KUKA KRL program: EPS_2_25369_MH2A_A_20251215023754.src

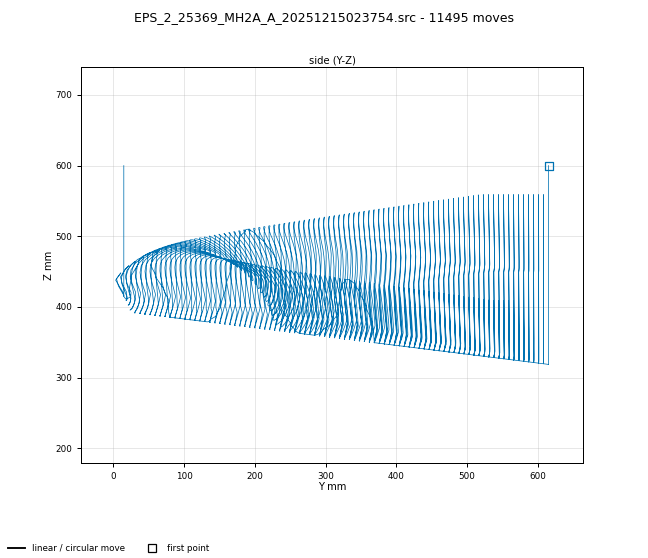
[picture p0: tool path of EPS_2_25369_MH2A_A_20251215023754.src, 11495 of 11497 moves have a stored position in this frame; points joined in program order, loops and branches not executed]
&ACCESS RVP
&REL 4
&COMMENT QRS 19112012
&PARAM EDITMASK = *
DEF PART()
EXT BAS (BAS_COMMAND :IN,REAL :IN )
INT I
BAS (#INITMOV,0 )

;KUKA QRS Post kuka4.cps  Date:22-06-2017 !

File_ID=2955

QRS_PRE_INIT()

;Init var - Until changes are made in qrs_pre_init
Outlet_Square_prg=0
Inlet_1_Square_prg=0
Inlet_2_Square_prg=0
Inlet_3_Square_prg=0
Inlet_4_Square_prg=0
Inlet_5_Square_prg=0

Outlet_1={X 0.000, Y 520.860, Z 458.500, B 0.000, E1 0.000 }
Inlet_1={X 0.000, Y 535.350, Z 258.500, B 0.000, E1 242.000 }
Outlet_1_type=201
Inlet_1_type=201
;QRS#1=Sidecore dimensions
;QRS#2=200-8" PVC SDR 35
;QRS#3=200-8" PVC SDR 35
;QRS#4=
;QRS#5=
;QRS#6=
;QRS#7=
;QRS#8=
;QRS#9=12-08 PSX
;QRS#10=12-08 PSX
;QRS#11=
;QRS#12=
;QRS#13=
;QRS#14=
;QRS#15=
;QRS#16=1220x127x838 2,75'
;QRS#17=EPS Height
;QRS#18=559
;QRS#19=*
;QRS#20= UPDATED VERSION 22-06-2017
;QRS#21=*
Outlet_Square=0100
Inlet_1_Square=0100
Inlet_2_Square=0
Inlet_3_Square=0
Inlet_4_Square=0
Inlet_5_Square=0
Mill_Square=1
Outlet_Square_Prg=204
Inlet_1_Square_prg=204

QRS_INIT()

$ADVANCE=5

; T1
PTP {E1 173.589,E2 173.589}
PTP {X 0,Y 615.517,A -85,B 0,C 180,E1 173.589,E2 173.589,E3 0,E4 0,E5 0,E6 0}
QRS_SPEED_INIT()
LIN {X 0,Y 615.517,Z 600,A -85,B 0,C 180,E1 173.589,E2 173.589,E3 0,E4 0,E5 0,E6 0} C_VEL
LIN {X 0,Y 615.517,Z 328.868,A -85,B 0,C 180,E1 173.589,E2 173.589} C_VEL
LIN {X 0,Y 615.517,Z 320.697,A -85,B 0,C 180,E1 173.589,E2 173.589} C_VEL
LIN {X 0,Y 615.495,Z 318.697,A -85,B 0,C 180,E1 173.403,E2 173.403} C_VEL
LIN {X 0,Y 615.469,Z 318.691,A -85,B 0,C 180,E1 170.801,E2 170.801} C_VEL
LIN {X 0,Y 615.46,Z 318.69,A -85,B 0,C 180,E1 168.139,E2 168.139} C_VEL
LIN {X 0,Y 615.493,Z 318.7,A -85,B 0,C 180,E1 165.451,E2 165.451} C_VEL
LIN {X 0,Y 615.461,Z 318.69,A -85,B 0,C 180,E1 162.729,E2 162.729} C_VEL
LIN {X 0,Y 615.458,Z 318.69,A -85,B 0,C 180,E1 160.661,E2 160.661} C_VEL
LIN {X 0,Y 615.457,Z 318.689,A -85,B 0,C 180,E1 158.567,E2 158.567} C_VEL
LIN {X 0,Y 615.486,Z 318.689,A -85,B 0,C 180,E1 155.989,E2 155.989} C_VEL
LIN {X 0,Y 615.489,Z 318.702,A -85,B 0,C 180,E1 153.556,E2 153.556} C_VEL
LIN {X 0,Y 615.491,Z 318.693,A -85,B 0,C 180,E1 151.342,E2 151.342} C_VEL
LIN {X 0,Y 615.465,Z 318.689,A -85,B 0,C 180,E1 148.915,E2 148.915} C_VEL
LIN {X 0,Y 615.466,Z 318.688,A -85,B 0,C 180,E1 146.467,E2 146.467} C_VEL
LIN {X 0,Y 615.494,Z 318.697,A -85,B 0,C 180,E1 143.576,E2 143.576} C_VEL
LIN {X 0,Y 615.464,Z 318.689,A -85,B 0,C 180,E1 140.939,E2 140.939} C_VEL
LIN {X 0,Y 615.471,Z 318.687,A -85,B 0,C 180,E1 138.525,E2 138.525} C_VEL
LIN {X 0,Y 615.499,Z 318.699,A -85,B 0,C 180,E1 135.851,E2 135.851} C_VEL
LIN {X 0,Y 615.467,Z 318.688,A -85,B 0,C 180,E1 133.045,E2 133.045} C_VEL
LIN {X 0,Y 615.476,Z 318.687,A -85,B 0,C 180,E1 130.606,E2 130.606} C_VEL
LIN {X 0,Y 615.491,Z 318.699,A -85,B 0,C 180,E1 128.012,E2 128.012} C_VEL
LIN {X 0,Y 615.497,Z 318.689,A -85,B 0,C 180,E1 125.614,E2 125.614} C_VEL
LIN {X 0,Y 615.472,Z 318.687,A -85,B 0,C 180,E1 123.236,E2 123.236} C_VEL
LIN {X 0,Y 615.471,Z 318.686,A -85,B 0,C 180,E1 120.92,E2 120.92} C_VEL
LIN {X 0,Y 615.495,Z 318.688,A -85,B 0,C 180,E1 118.451,E2 118.451} C_VEL
LIN {X 0,Y 615.486,Z 318.687,A -85,B 0,C 180,E1 115.568,E2 115.568} C_VEL
LIN {X 0,Y 615.479,Z 318.686,A -85,B 0,C 180,E1 112.844,E2 112.844} C_VEL
LIN {X 0,Y 615.497,Z 318.695,A -85,B 0,C 180,E1 110.032,E2 110.032} C_VEL
LIN {X 0,Y 615.473,Z 318.686,A -85,B 0,C 180,E1 107.27,E2 107.27} C_VEL
LIN {X 0,Y 615.494,Z 318.691,A -85,B 0,C 180,E1 104.549,E2 104.549} C_VEL
LIN {X 0,Y 615.49,Z 318.689,A -85,B 0,C 180,E1 101.86,E2 101.86} C_VEL
LIN {X 0,Y 615.478,Z 318.685,A -85,B 0,C 180,E1 99.199,E2 99.199} C_VEL
LIN {X 0,Y 615.494,Z 318.694,A -85,B 0,C 180,E1 96.556,E2 96.556} C_VEL
LIN {X 0,Y 615.489,Z 318.688,A -85,B 0,C 180,E1 93.928,E2 93.928} C_VEL
LIN {X 0,Y 615.48,Z 318.684,A -85,B 0,C 180,E1 91.309,E2 91.309} C_VEL
LIN {X 0,Y 615.494,Z 318.694,A -85,B 0,C 180,E1 88.691,E2 88.691} C_VEL
LIN {X 0,Y 615.491,Z 318.688,A -85,B 0,C 180,E1 86.072,E2 86.072} C_VEL
LIN {X 0,Y 615.48,Z 318.684,A -85,B 0,C 180,E1 83.43,E2 83.43} C_VEL
LIN {X 0,Y 615.49,Z 318.695,A -85,B 0,C 180,E1 80.801,E2 80.801} C_VEL
LIN {X 0,Y 615.49,Z 318.687,A -85,B 0,C 180,E1 78.14,E2 78.14} C_VEL
LIN {X 0,Y 615.484,Z 318.684,A -85,B 0,C 180,E1 75.451,E2 75.451} C_VEL
LIN {X 0,Y 615.498,Z 318.699,A -85,B 0,C 180,E1 72.73,E2 72.73} C_VEL
LIN {X 0,Y 615.485,Z 318.684,A -85,B 0,C 180,E1 69.968,E2 69.968} C_VEL
LIN {X 0,Y 615.491,Z 318.69,A -85,B 0,C 180,E1 67.156,E2 67.156} C_VEL
LIN {X 0,Y 615.5,Z 318.684,A -85,B 0,C 180,E1 64.286,E2 64.286} C_VEL
LIN {X 0,Y 615.493,Z 318.683,A -85,B 0,C 180,E1 61.549,E2 61.549} C_VEL
LIN {X 0,Y 615.491,Z 318.702,A -85,B 0,C 180,E1 58.914,E2 58.914} C_VEL
LIN {X 0,Y 615.491,Z 318.688,A -85,B 0,C 180,E1 56.466,E2 56.466} C_VEL
LIN {X 0,Y 615.489,Z 318.685,A -85,B 0,C 180,E1 53.576,E2 53.576} C_VEL
LIN {X 0,Y 615.492,Z 318.699,A -85,B 0,C 180,E1 50.938,E2 50.938} C_VEL
LIN {X 0,Y 615.495,Z 318.686,A -85,B 0,C 180,E1 48.528,E2 48.528} C_VEL
LIN {X 0,Y 615.493,Z 318.682,A -85,B 0,C 180,E1 45.852,E2 45.852} C_VEL
LIN {X 0,Y 615.492,Z 318.699,A -85,B 0,C 180,E1 43.049,E2 43.049} C_VEL
LIN {X 0,Y 615.495,Z 318.685,A -85,B 0,C 180,E1 40.606,E2 40.606} C_VEL
LIN {X 0,Y 615.492,Z 318.789,A -85,B 0,C 180,E1 39.236,E2 39.236} C_VEL
LIN {X 0,Y 615.494,Z 331.581,A -85,B 0,C 180,E1 38.799,E2 38.799} C_VEL
LIN {X 0,Y 615.494,Z 341.036,A -85,B 0,C 180,E1 38.38,E2 38.38} C_VEL
LIN {X 0,Y 615.496,Z 349.628,A -85,B 0,C 180,E1 37.918,E2 37.918} C_VEL
LIN {X 0,Y 615.498,Z 358.544,A -85,B 0,C 180,E1 37.338,E2 37.338} C_VEL
LIN {X 0,Y 615.499,Z 366.968,A -85,B 0,C 180,E1 36.681,E2 36.681} C_VEL
LIN {X 0,Y 615.497,Z 374.514,A -85,B 0,C 180,E1 35.984,E2 35.984} C_VEL
LIN {X 0,Y 615.498,Z 381.527,A -85,B 0,C 180,E1 35.214,E2 35.214} C_VEL
LIN {X 0,Y 615.496,Z 386.825,A -85,B 0,C 180,E1 34.532,E2 34.532} C_VEL
LIN {X 0,Y 615.491,Z 391.828,A -85,B 0,C 180,E1 33.78,E2 33.78} C_VEL
LIN {X 0,Y 615.493,Z 396.922,A -85,B 0,C 180,E1 32.846,E2 32.846} C_VEL
LIN {X 0,Y 615.492,Z 400.615,A -85,B 0,C 180,E1 32.009,E2 32.009} C_VEL
LIN {X 0,Y 615.488,Z 404.238,A -85,B 0,C 180,E1 30.92,E2 30.92} C_VEL
LIN {X 0,Y 615.493,Z 406.751,A -85,B 0,C 180,E1 29.798,E2 29.798} C_VEL
LIN {X 0,Y 615.485,Z 407.427,A -85,B 0,C 180,E1 29.406,E2 29.406} C_VEL
LIN {X 0,Y 615.497,Z 408.272,A -85,B 0,C 180,E1 28.455,E2 28.455} C_VEL
LIN {X 0,Y 615.489,Z 407.929,A -85,B 0,C 180,E1 27.048,E2 27.048} C_VEL
LIN {X 0,Y 615.489,Z 407.306,A -85,B 0,C 180,E1 26.444,E2 26.444} C_VEL
LIN {X 0,Y 615.489,Z 405.769,A -85,B 0,C 180,E1 25.572,E2 25.572} C_VEL
LIN {X 0,Y 615.496,Z 403.25,A -85,B 0,C 180,E1 24.631,E2 24.631} C_VEL
LIN {X 0,Y 615.486,Z 399.206,A -85,B 0,C 180,E1 23.556,E2 23.556} C_VEL
LIN {X 0,Y 615.498,Z 394.51,A -85,B 0,C 180,E1 22.597,E2 22.597} C_VEL
LIN {X 0,Y 615.496,Z 389.635,A -85,B 0,C 180,E1 21.783,E2 21.783} C_VEL
LIN {X 0,Y 615.496,Z 383.247,A -85,B 0,C 180,E1 20.905,E2 20.905} C_VEL
LIN {X 0,Y 615.499,Z 376.823,A -85,B 0,C 180,E1 20.165,E2 20.165} C_VEL
LIN {X 0,Y 615.499,Z 370.184,A -85,B 0,C 180,E1 19.511,E2 19.511} C_VEL
LIN {X 0,Y 615.498,Z 361.856,A -85,B 0,C 180,E1 18.818,E2 18.818} C_VEL
LIN {X 0,Y 615.497,Z 352.996,A -85,B 0,C 180,E1 18.202,E2 18.202} C_VEL
LIN {X 0,Y 615.497,Z 344.313,A -85,B 0,C 180,E1 17.699,E2 17.699} C_VEL
LIN {X 0,Y 615.498,Z 335.372,A -85,B 0,C 180,E1 17.27,E2 17.27} C_VEL
LIN {X 0,Y 615.497,Z 326.627,A -85,B 0,C 180,E1 16.928,E2 16.928} C_VEL
LIN {X 0,Y 615.497,Z 319.573,A -85,B 0,C 180,E1 16.672,E2 16.672} C_VEL
LIN {X 0,Y 615.495,Z 318.786,A -85,B 0,C 180,E1 16.512,E2 16.512} C_VEL
LIN {X 0,Y 615.463,Z 318.69,A -85,B 0,C 180,E1 13.875,E2 13.875} C_VEL
LIN {X 0,Y 615.468,Z 318.69,A -85,B 0,C 180,E1 11.193,E2 11.193} C_VEL
LIN {X 0,Y 615.496,Z 318.698,A -85,B 0,C 180,E1 8.537,E2 8.537} C_VEL
LIN {X 0,Y 615.456,Z 318.691,A -85,B 0,C 180,E1 5.899,E2 5.899} C_VEL
LIN {X 0,Y 615.467,Z 318.69,A -85,B 0,C 180,E1 3.273,E2 3.273} C_VEL
LIN {X 0,Y 615.496,Z 318.699,A -85,B 0,C 180,E1 0.654,E2 0.654} C_VEL
LIN {X 0,Y 615.455,Z 318.692,A -85,B 0,C 180,E1 -1.963,E2 -1.963} C_VEL
LIN {X 0,Y 615.452,Z 318.692,A -85,B 0,C 180,E1 -3.929,E2 -3.929} C_VEL
LIN {X 0,Y 615.454,Z 318.692,A -85,B 0,C 180,E1 -5.899,E2 -5.899} C_VEL
LIN {X 0,Y 615.451,Z 318.693,A -85,B 0,C 180,E1 -7.876,E2 -7.876} C_VEL
LIN {X 0,Y 615.451,Z 318.692,A -85,B 0,C 180,E1 -9.863,E2 -9.863} C_VEL
LIN {X 0,Y 615.449,Z 318.693,A -85,B 0,C 180,E1 -11.862,E2 -11.862} C_VEL
LIN {X 0,Y 615.445,Z 318.693,A -85,B 0,C 180,E1 -13.923,E2 -13.923} C_VEL
LIN {X 0,Y 615.472,Z 318.691,A -85,B 0,C 180,E1 -16.587,E2 -16.587} C_VEL
LIN {X 0,Y 615.479,Z 318.694,A -85,B 0,C 180,E1 -19.338,E2 -19.338} C_VEL
LIN {X 0,Y 615.461,Z 318.695,A -85,B 0,C 180,E1 -21.433,E2 -21.433} C_VEL
LIN {X 0,Y 615.452,Z 318.694,A -85,B 0,C 180,E1 -23.558,E2 -23.558} C_VEL
LIN {X 0,Y 615.441,Z 318.694,A -85,B 0,C 180,E1 -25.718,E2 -25.718} C_VEL
LIN {X 0,Y 615.438,Z 318.693,A -85,B 0,C 180,E1 -27.918,E2 -27.918} C_VEL
LIN {X 0,Y 615.492,Z 318.701,A -85,B 0,C 180,E1 -30.92,E2 -30.92} C_VEL
LIN {X 0,Y 615.442,Z 318.695,A -85,B 0,C 180,E1 -33.53,E2 -33.53} C_VEL
LIN {X 0,Y 615.435,Z 318.694,A -85,B 0,C 180,E1 -35.829,E2 -35.829} C_VEL
LIN {X 0,Y 615.445,Z 318.694,A -85,B 0,C 180,E1 -38.072,E2 -38.072} C_VEL
LIN {X 0,Y 615.491,Z 318.696,A -85,B 0,C 180,E1 -40.606,E2 -40.606} C_VEL
LIN {X 0,Y 615.446,Z 318.696,A -85,B 0,C 180,E1 -43.248,E2 -43.248} C_VEL
LIN {X 0,Y 615.445,Z 318.694,A -85,B 0,C 180,E1 -46.007,E2 -46.007} C_VEL
LIN {X 0,Y 615.469,Z 318.698,A -85,B 0,C 180,E1 -48.908,E2 -48.908} C_VEL
LIN {X 0,Y 615.446,Z 318.698,A -85,B 0,C 180,E1 -51.094,E2 -51.094} C_VEL
LIN {X 0,Y 615.427,Z 318.696,A -85,B 0,C 180,E1 -53.572,E2 -53.572} C_VEL
LIN {X 0,Y 615.495,Z 318.898,A -85,B 0,C 180,E1 -54.687,E2 -54.687} C_VEL
LIN {X 0,Y 615.497,Z 333.444,A -85,B 0,C 180,E1 -57.35,E2 -57.35} C_VEL
LIN {X 0,Y 615.496,Z 348.208,A -85,B 0,C 180,E1 -60.204,E2 -60.204} C_VEL
LIN {X 0,Y 615.465,Z 362.707,A -85,B 0,C 180,E1 -62.96,E2 -62.96} C_VEL
LIN {X 0,Y 615.477,Z 375.666,A -85,B 0,C 180,E1 -65.369,E2 -65.369} C_VEL
LIN {X 0,Y 615.496,Z 391.293,A -85,B 0,C 180,E1 -68.217,E2 -68.217} C_VEL
LIN {X 0,Y 615.462,Z 406.91,A -85,B 0,C 180,E1 -71.008,E2 -71.008} C_VEL
LIN {X 0,Y 615.462,Z 421.502,A -85,B 0,C 180,E1 -73.578,E2 -73.578} C_VEL
LIN {X 0,Y 615.488,Z 438.093,A -85,B 0,C 180,E1 -76.463,E2 -76.463} C_VEL
LIN {X 0,Y 615.485,Z 448.706,A -85,B 0,C 180,E1 -78.265,E2 -78.265} C_VEL
LIN {X 0,Y 615.482,Z 449.705,A -85,B 0,C 180,E1 -78.327,E2 -78.327} C_VEL
LIN {X 0,Y 615.47,Z 464.052,A -85,B 0,C 180,E1 -78.598,E2 -78.598} C_VEL
LIN {X 0,Y 615.474,Z 476.487,A -85,B 0,C 180,E1 -78.961,E2 -78.961} C_VEL
LIN {X 0,Y 615.494,Z 487.108,A -85,B 0,C 180,E1 -79.384,E2 -79.384} C_VEL
LIN {X 0,Y 615.497,Z 498.603,A -85,B 0,C 180,E1 -79.972,E2 -79.972} C_VEL
LIN {X 0,Y 615.499,Z 510.015,A -85,B 0,C 180,E1 -80.719,E2 -80.719} C_VEL
LIN {X 0,Y 615.498,Z 519.243,A -85,B 0,C 180,E1 -81.464,E2 -81.464} C_VEL
LIN {X 0,Y 615.499,Z 527.669,A -85,B 0,C 180,E1 -82.29,E2 -82.29} C_VEL
LIN {X 0,Y 615.498,Z 535.689,A -85,B 0,C 180,E1 -83.258,E2 -83.258} C_VEL
LIN {X 0,Y 615.499,Z 541.428,A -85,B 0,C 180,E1 -84.102,E2 -84.102} C_VEL
LIN {X 0,Y 615.495,Z 546.876,A -85,B 0,C 180,E1 -85.087,E2 -85.087} C_VEL
LIN {X 0,Y 615.497,Z 551.143,A -85,B 0,C 180,E1 -86.072,E2 -86.072} C_VEL
LIN {X 0,Y 615.494,Z 553.397,A -85,B 0,C 180,E1 -86.727,E2 -86.727} C_VEL
LIN {X 0,Y 615.496,Z 555.231,A -85,B 0,C 180,E1 -87.382,E2 -87.382} C_VEL
LIN {X 0,Y 615.5,Z 556.61,A -85,B 0,C 180,E1 -88.037,E2 -88.037} C_VEL
LIN {X 0,Y 615.496,Z 558.173,A -85,B 0,C 180,E1 -89.346,E2 -89.346} C_VEL
LIN {X 0,Y 615.494,Z 558.389,A -85,B 0,C 180,E1 -90,E2 -90} C_VEL
LIN {X 0,Y 615.495,Z 557.581,A -85,B 0,C 180,E1 -91.309,E2 -91.309} C_VEL
LIN {X 0,Y 615.5,Z 556.61,A -85,B 0,C 180,E1 -91.963,E2 -91.963} C_VEL
LIN {X 0,Y 615.496,Z 555.231,A -85,B 0,C 180,E1 -92.618,E2 -92.618} C_VEL
LIN {X 0,Y 615.495,Z 552.352,A -85,B 0,C 180,E1 -93.601,E2 -93.601} C_VEL
LIN {X 0,Y 615.497,Z 548.448,A -85,B 0,C 180,E1 -94.584,E2 -94.584} C_VEL
LIN {X 0,Y 615.499,Z 543.41,A -85,B 0,C 180,E1 -95.57,E2 -95.57} C_VEL
LIN {X 0,Y 615.497,Z 536.856,A -85,B 0,C 180,E1 -96.584,E2 -96.584} C_VEL
LIN {X 0,Y 615.497,Z 529.134,A -85,B 0,C 180,E1 -97.545,E2 -97.545} C_VEL
LIN {X 0,Y 615.498,Z 521.055,A -85,B 0,C 180,E1 -98.371,E2 -98.371} C_VEL
LIN {X 0,Y 615.499,Z 511.154,A -85,B 0,C 180,E1 -99.198,E2 -99.198} C_VEL
LIN {X 0,Y 615.498,Z 499.986,A -85,B 0,C 180,E1 -99.945,E2 -99.945} C_VEL
LIN {X 0,Y 615.497,Z 489.05,A -85,B 0,C 180,E1 -100.526,E2 -100.526} C_VEL
LIN {X 0,Y 615.476,Z 477.622,A -85,B 0,C 180,E1 -101,E2 -101} C_VEL
LIN {X 0,Y 615.469,Z 465.798,A -85,B 0,C 180,E1 -101.36,E2 -101.36} C_VEL
LIN {X 0,Y 615.48,Z 452.013,A -85,B 0,C 180,E1 -101.631,E2 -101.631} C_VEL
LIN {X 0,Y 615.484,Z 449.247,A -85,B 0,C 180,E1 -101.693,E2 -101.693} C_VEL
LIN {X 0,Y 615.491,Z 447.83,A -85,B 0,C 180,E1 -101.86,E2 -101.86} C_VEL
LIN {X 0,Y 615.489,Z 432.252,A -85,B 0,C 180,E1 -104.549,E2 -104.549} C_VEL
LIN {X 0,Y 615.492,Z 416.659,A -85,B 0,C 180,E1 -107.27,E2 -107.27} C_VEL
LIN {X 0,Y 615.477,Z 401.055,A -85,B 0,C 180,E1 -110.033,E2 -110.033} C_VEL
LIN {X 0,Y 615.474,Z 386.808,A -85,B 0,C 180,E1 -112.595,E2 -112.595} C_VEL
LIN {X 0,Y 615.488,Z 372.144,A -85,B 0,C 180,E1 -115.281,E2 -115.281} C_VEL
LIN {X 0,Y 615.473,Z 356.66,A -85,B 0,C 180,E1 -118.181,E2 -118.181} C_VEL
LIN {X 0,Y 615.464,Z 344.37,A -85,B 0,C 180,E1 -120.54,E2 -120.54} C_VEL
LIN {X 0,Y 615.489,Z 330.389,A -85,B 0,C 180,E1 -123.235,E2 -123.235} C_VEL
LIN {X 0,Y 615.495,Z 319.029,A -85,B 0,C 180,E1 -125.413,E2 -125.413} C_VEL
LIN {X 0,Y 615.468,Z 318.698,A -85,B 0,C 180,E1 -125.831,E2 -125.831} C_VEL
LIN {X 0,Y 615.442,Z 318.697,A -85,B 0,C 180,E1 -128.071,E2 -128.071} C_VEL
LIN {X 0,Y 615.431,Z 318.695,A -85,B 0,C 180,E1 -130.61,E2 -130.61} C_VEL
LIN {X 0,Y 615.494,Z 318.694,A -85,B 0,C 180,E1 -133.243,E2 -133.243} C_VEL
LIN {X 0,Y 615.443,Z 318.696,A -85,B 0,C 180,E1 -136.005,E2 -136.005} C_VEL
LIN {X 0,Y 615.436,Z 318.695,A -85,B 0,C 180,E1 -138.522,E2 -138.522} C_VEL
LIN {X 0,Y 615.487,Z 318.694,A -85,B 0,C 180,E1 -141.095,E2 -141.095} C_VEL
LIN {X 0,Y 615.472,Z 318.697,A -85,B 0,C 180,E1 -143.574,E2 -143.574} C_VEL
LIN {X 0,Y 615.441,Z 318.695,A -85,B 0,C 180,E1 -145.975,E2 -145.975} C_VEL
LIN {X 0,Y 615.438,Z 318.694,A -85,B 0,C 180,E1 -148.312,E2 -148.312} C_VEL
LIN {X 0,Y 615.454,Z 318.693,A -85,B 0,C 180,E1 -150.592,E2 -150.592} C_VEL
LIN {X 0,Y 615.467,Z 318.695,A -85,B 0,C 180,E1 -153.555,E2 -153.555} C_VEL
LIN {X 0,Y 615.44,Z 318.693,A -85,B 0,C 180,E1 -155.998,E2 -155.998} C_VEL
LIN {X 0,Y 615.442,Z 318.694,A -85,B 0,C 180,E1 -157.862,E2 -157.862} C_VEL
LIN {X 0,Y 615.439,Z 318.694,A -85,B 0,C 180,E1 -159.965,E2 -159.965} C_VEL
LIN {X 0,Y 615.488,Z 318.692,A -85,B 0,C 180,E1 -162.729,E2 -162.729} C_VEL
LIN {X 0,Y 615.467,Z 318.694,A -85,B 0,C 180,E1 -165.45,E2 -165.45} C_VEL
LIN {X 0,Y 615.463,Z 318.693,A -85,B 0,C 180,E1 -167.469,E2 -167.469} C_VEL
LIN {X 0,Y 615.461,Z 318.693,A -85,B 0,C 180,E1 -169.473,E2 -169.473} C_VEL
LIN {X 0,Y 615.457,Z 318.694,A -85,B 0,C 180,E1 -171.463,E2 -171.463} C_VEL
LIN {X 0,Y 615.461,Z 318.693,A -85,B 0,C 180,E1 -173.443,E2 -173.443} C_VEL
LIN {X 0,Y 615.458,Z 318.693,A -85,B 0,C 180,E1 -175.415,E2 -175.415} C_VEL
LIN {X 0,Y 615.463,Z 318.692,A -85,B 0,C 180,E1 -177.382,E2 -177.382} C_VEL
LIN {X 0,Y 615.455,Z 318.691,A -85,B 0,C 180,E1 -180,E2 -180} C_VEL
LIN {X 0,Y 615.495,Z 318.696,A -85,B 0,C 180,E1 -182.618,E2 -182.618} C_VEL
LIN {X 0,Y 615.468,Z 318.692,A -85,B 0,C 180,E1 -185.241,E2 -185.241} C_VEL
LIN {X 0,Y 615.495,Z 318.697,A -85,B 0,C 180,E1 -186.597,E2 -186.597} C_VEL
LIN {X 0,Y 614.802,Z 318.837,A -85,B 0,C 180,E1 -187.142,E2 -187.142} C_VEL
LIN {X 0,Y 611.956,Z 319.252,A -85,B 0,C 180,E1 -188.028,E2 -188.028} C_VEL
LIN {X 0,Y 609.563,Z 319.562,A -85,B 0,C 180,E1 -188.741,E2 -188.741} C_VEL
LIN {X 0,Y 608.529,Z 319.68,A -85,B 0,C 180,E1 -189.29,E2 -189.29} C_VEL
LIN {X 0,Y 608.439,Z 319.689,A -85,B 0,C 180,E1 -189.476,E2 -189.476} C_VEL
LIN {X 0,Y 608.444,Z 319.69,A -85,B 0,C 180,E1 -192,E2 -192} C_VEL
LIN {X 0,Y 608.471,Z 319.694,A -85,B 0,C 180,E1 -194.721,E2 -194.721} C_VEL
LIN {X 0,Y 608.431,Z 319.69,A -85,B 0,C 180,E1 -197.477,E2 -197.477} C_VEL
LIN {X 0,Y 608.434,Z 319.69,A -85,B 0,C 180,E1 -199.571,E2 -199.571} C_VEL
LIN {X 0,Y 608.454,Z 319.687,A -85,B 0,C 180,E1 -201.692,E2 -201.692} C_VEL
LIN {X 0,Y 608.45,Z 319.696,A -85,B 0,C 180,E1 -204.571,E2 -204.571} C_VEL
LIN {X 0,Y 608.436,Z 319.689,A -85,B 0,C 180,E1 -207.519,E2 -207.519} C_VEL
LIN {X 0,Y 608.464,Z 319.69,A -85,B 0,C 180,E1 -209.973,E2 -209.973} C_VEL
LIN {X 0,Y 608.448,Z 319.69,A -85,B 0,C 180,E1 -212.88,E2 -212.88} C_VEL
LIN {X 0,Y 608.431,Z 319.69,A -85,B 0,C 180,E1 -215.279,E2 -215.279} C_VEL
LIN {X 0,Y 608.469,Z 319.696,A -85,B 0,C 180,E1 -218.242,E2 -218.242} C_VEL
LIN {X 0,Y 608.433,Z 319.69,A -85,B 0,C 180,E1 -221.179,E2 -221.179} C_VEL
LIN {X 0,Y 608.475,Z 319.69,A -85,B 0,C 180,E1 -223.869,E2 -223.869} C_VEL
LIN {X 0,Y 608.465,Z 319.688,A -85,B 0,C 180,E1 -226.692,E2 -226.692} C_VEL
LIN {X 0,Y 608.443,Z 319.689,A -85,B 0,C 180,E1 -228.824,E2 -228.824} C_VEL
LIN {X 0,Y 608.468,Z 319.691,A -85,B 0,C 180,E1 -231.76,E2 -231.76} C_VEL
LIN {X 0,Y 608.443,Z 319.69,A -85,B 0,C 180,E1 -234.723,E2 -234.723} C_VEL
LIN {X 0,Y 608.467,Z 319.688,A -85,B 0,C 180,E1 -237.477,E2 -237.477} C_VEL
LIN {X 0,Y 608.48,Z 319.69,A -85,B 0,C 180,E1 -240.222,E2 -240.222} C_VEL
LIN {X 0,Y 608.467,Z 319.686,A -85,B 0,C 180,E1 -242.795,E2 -242.795} C_VEL
LIN {X 0,Y 608.453,Z 319.69,A -85,B 0,C 180,E1 -245.43,E2 -245.43} C_VEL
LIN {X 0,Y 608.467,Z 319.689,A -85,B 0,C 180,E1 -248.309,E2 -248.309} C_VEL
LIN {X 0,Y 608.456,Z 319.688,A -85,B 0,C 180,E1 -251.131,E2 -251.131} C_VEL
LIN {X 0,Y 608.467,Z 319.694,A -85,B 0,C 180,E1 -253.907,E2 -253.907} C_VEL
LIN {X 0,Y 608.459,Z 319.687,A -85,B 0,C 180,E1 -256.644,E2 -256.644} C_VEL
LIN {X 0,Y 608.47,Z 319.69,A -85,B 0,C 180,E1 -259.351,E2 -259.351} C_VEL
LIN {X 0,Y 608.481,Z 319.688,A -85,B 0,C 180,E1 -262.033,E2 -262.033} C_VEL
LIN {X 0,Y 608.461,Z 319.686,A -85,B 0,C 180,E1 -264.698,E2 -264.698} C_VEL
LIN {X 0,Y 608.484,Z 319.69,A -85,B 0,C 180,E1 -267.352,E2 -267.352} C_VEL
LIN {X 0,Y 608.481,Z 319.687,A -85,B 0,C 180,E1 -270,E2 -270} C_VEL
LIN {X 0,Y 608.472,Z 319.685,A -85,B 0,C 180,E1 -272.648,E2 -272.648} C_VEL
LIN {X 0,Y 608.473,Z 319.693,A -85,B 0,C 180,E1 -275.302,E2 -275.302} C_VEL
LIN {X 0,Y 608.481,Z 319.686,A -85,B 0,C 180,E1 -277.967,E2 -277.967} C_VEL
LIN {X 0,Y 608.463,Z 319.687,A -85,B 0,C 180,E1 -280.65,E2 -280.65} C_VEL
LIN {X 0,Y 608.472,Z 319.696,A -85,B 0,C 180,E1 -283.356,E2 -283.356} C_VEL
LIN {X 0,Y 608.461,Z 319.687,A -85,B 0,C 180,E1 -286.093,E2 -286.093} C_VEL
LIN {X 0,Y 608.459,Z 319.69,A -85,B 0,C 180,E1 -288.869,E2 -288.869} C_VEL
LIN {X 0,Y 608.472,Z 319.688,A -85,B 0,C 180,E1 -291.691,E2 -291.691} C_VEL
LIN {X 0,Y 608.455,Z 319.689,A -85,B 0,C 180,E1 -294.57,E2 -294.57} C_VEL
LIN {X 0,Y 608.485,Z 319.693,A -85,B 0,C 180,E1 -297.208,E2 -297.208} C_VEL
LIN {X 0,Y 608.469,Z 319.685,A -85,B 0,C 180,E1 -299.971,E2 -299.971} C_VEL
LIN {X 0,Y 608.467,Z 319.688,A -85,B 0,C 180,E1 -302.523,E2 -302.523} C_VEL
LIN {X 0,Y 608.451,Z 319.694,A -85,B 0,C 180,E1 -305.276,E2 -305.276} C_VEL
LIN {X 0,Y 608.471,Z 319.686,A -85,B 0,C 180,E1 -307.745,E2 -307.745} C_VEL
LIN {X 0,Y 608.478,Z 319.686,A -85,B 0,C 180,E1 -310.332,E2 -310.332} C_VEL
LIN {X 0,Y 608.479,Z 319.689,A -85,B 0,C 180,E1 -313.309,E2 -313.309} C_VEL
LIN {X 0,Y 608.472,Z 319.686,A -85,B 0,C 180,E1 -316.131,E2 -316.131} C_VEL
LIN {X 0,Y 608.46,Z 319.697,A -85,B 0,C 180,E1 -318.824,E2 -318.824} C_VEL
LIN {X 0,Y 608.488,Z 319.875,A -85,B 0,C 180,E1 -320.661,E2 -320.661} C_VEL
LIN {X 0,Y 608.513,Z 332.249,A -85,B 0,C 180,E1 -321.097,E2 -321.097} C_VEL
LIN {X 0,Y 608.506,Z 341.54,A -85,B 0,C 180,E1 -321.516,E2 -321.516} C_VEL
LIN {X 0,Y 608.498,Z 351.312,A -85,B 0,C 180,E1 -322.06,E2 -322.06} C_VEL
LIN {X 0,Y 608.491,Z 359.545,A -85,B 0,C 180,E1 -322.61,E2 -322.61} C_VEL
LIN {X 0,Y 608.471,Z 368.109,A -85,B 0,C 180,E1 -323.293,E2 -323.293} C_VEL
LIN {X 0,Y 608.473,Z 375.088,A -85,B 0,C 180,E1 -323.949,E2 -323.949} C_VEL
LIN {X 0,Y 608.462,Z 382.076,A -85,B 0,C 180,E1 -324.723,E2 -324.723} C_VEL
LIN {X 0,Y 608.461,Z 388.204,A -85,B 0,C 180,E1 -325.53,E2 -325.53} C_VEL
LIN {X 0,Y 608.457,Z 393.298,A -85,B 0,C 180,E1 -326.329,E2 -326.329} C_VEL
LIN {X 0,Y 608.428,Z 397.518,A -85,B 0,C 180,E1 -327.119,E2 -327.119} C_VEL
LIN {X 0,Y 608.423,Z 402.432,A -85,B 0,C 180,E1 -328.293,E2 -328.293} C_VEL
LIN {X 0,Y 608.443,Z 403.951,A -85,B 0,C 180,E1 -328.731,E2 -328.731} C_VEL
LIN {X 0,Y 608.425,Z 405.914,A -85,B 0,C 180,E1 -329.453,E2 -329.453} C_VEL
LIN {X 0,Y 608.442,Z 407.417,A -85,B 0,C 180,E1 -330.219,E2 -330.219} C_VEL
LIN {X 0,Y 608.421,Z 408.78,A -85,B 0,C 180,E1 -331.386,E2 -331.386} C_VEL
LIN {X 0,Y 608.42,Z 408.912,A -85,B 0,C 180,E1 -332.481,E2 -332.481} C_VEL
LIN {X 0,Y 608.42,Z 408.331,A -85,B 0,C 180,E1 -333.224,E2 -333.224} C_VEL
LIN {X 0,Y 608.421,Z 406.712,A -85,B 0,C 180,E1 -334.286,E2 -334.286} C_VEL
LIN {X 0,Y 608.425,Z 403.735,A -85,B 0,C 180,E1 -335.428,E2 -335.428} C_VEL
LIN {X 0,Y 608.443,Z 399.625,A -85,B 0,C 180,E1 -336.515,E2 -336.515} C_VEL
LIN {X 0,Y 608.447,Z 394.655,A -85,B 0,C 180,E1 -337.523,E2 -337.523} C_VEL
LIN {X 0,Y 608.462,Z 388.713,A -85,B 0,C 180,E1 -338.486,E2 -338.486} C_VEL
LIN {X 0,Y 608.472,Z 382.488,A -85,B 0,C 180,E1 -339.317,E2 -339.317} C_VEL
LIN {X 0,Y 608.465,Z 375.703,A -85,B 0,C 180,E1 -340.078,E2 -340.078} C_VEL
LIN {X 0,Y 608.467,Z 366.351,A -85,B 0,C 180,E1 -340.956,E2 -340.956} C_VEL
LIN {X 0,Y 608.515,Z 355.759,A -85,B 0,C 180,E1 -341.747,E2 -341.747} C_VEL
LIN {X 0,Y 608.499,Z 345.79,A -85,B 0,C 180,E1 -342.351,E2 -342.351} C_VEL
LIN {X 0,Y 608.513,Z 336.117,A -85,B 0,C 180,E1 -342.828,E2 -342.828} C_VEL
LIN {X 0,Y 608.541,Z 326.217,A -85,B 0,C 180,E1 -343.218,E2 -343.218} C_VEL
LIN {X 0,Y 608.552,Z 320.356,A -85,B 0,C 180,E1 -343.439,E2 -343.439} C_VEL
LIN {X 0,Y 608.495,Z 319.76,A -85,B 0,C 180,E1 -343.57,E2 -343.57} C_VEL
LIN {X 0,Y 608.461,Z 319.689,A -85,B 0,C 180,E1 -345.981,E2 -345.981} C_VEL
LIN {X 0,Y 608.459,Z 319.687,A -85,B 0,C 180,E1 -348.676,E2 -348.676} C_VEL
LIN {X 0,Y 608.46,Z 319.697,A -85,B 0,C 180,E1 -351.364,E2 -351.364} C_VEL
LIN {X 0,Y 608.435,Z 319.691,A -85,B 0,C 180,E1 -354.033,E2 -354.033} C_VEL
LIN {X 0,Y 608.46,Z 319.688,A -85,B 0,C 180,E1 -356.689,E2 -356.689} C_VEL
LIN {X 0,Y 608.487,Z 319.693,A -85,B 0,C 180,E1 -359.338,E2 -359.338} C_VEL
LIN {X 0,Y 608.425,Z 319.692,A -85,B 0,C 180,E1 -361.986,E2 -361.986} C_VEL
LIN {X 0,Y 608.422,Z 319.692,A -85,B 0,C 180,E1 -363.974,E2 -363.974} C_VEL
LIN {X 0,Y 608.447,Z 319.69,A -85,B 0,C 180,E1 -366.633,E2 -366.633} C_VEL
LIN {X 0,Y 608.471,Z 319.693,A -85,B 0,C 180,E1 -369.306,E2 -369.306} C_VEL
LIN {X 0,Y 608.431,Z 319.69,A -85,B 0,C 180,E1 -372,E2 -372} C_VEL
LIN {X 0,Y 608.462,Z 319.691,A -85,B 0,C 180,E1 -374.721,E2 -374.721} C_VEL
LIN {X 0,Y 608.441,Z 319.692,A -85,B 0,C 180,E1 -377.477,E2 -377.477} C_VEL
LIN {X 0,Y 608.432,Z 319.692,A -85,B 0,C 180,E1 -379.571,E2 -379.571} C_VEL
LIN {X 0,Y 608.438,Z 319.69,A -85,B 0,C 180,E1 -381.693,E2 -381.693} C_VEL
LIN {X 0,Y 608.439,Z 319.693,A -85,B 0,C 180,E1 -384.572,E2 -384.572} C_VEL
LIN {X 0,Y 608.428,Z 319.692,A -85,B 0,C 180,E1 -387.519,E2 -387.519} C_VEL
LIN {X 0,Y 608.424,Z 319.691,A -85,B 0,C 180,E1 -389.967,E2 -389.967} C_VEL
LIN {X 0,Y 608.442,Z 319.699,A -85,B 0,C 180,E1 -392.881,E2 -392.881} C_VEL
LIN {X 0,Y 608.42,Z 319.695,A -85,B 0,C 180,E1 -395.279,E2 -395.279} C_VEL
LIN {X 0,Y 608.433,Z 319.69,A -85,B 0,C 180,E1 -397.749,E2 -397.749} C_VEL
LIN {X 0,Y 608.432,Z 319.693,A -85,B 0,C 180,E1 -400.329,E2 -400.329} C_VEL
LIN {X 0,Y 608.438,Z 319.691,A -85,B 0,C 180,E1 -403.307,E2 -403.307} C_VEL
LIN {X 0,Y 608.439,Z 319.691,A -85,B 0,C 180,E1 -406.129,E2 -406.129} C_VEL
LIN {X 0,Y 608.444,Z 319.696,A -85,B 0,C 180,E1 -408.824,E2 -408.824} C_VEL
LIN {X 0,Y 608.401,Z 319.695,A -85,B 0,C 180,E1 -411.408,E2 -411.408} C_VEL
LIN {X 0,Y 608.433,Z 319.693,A -85,B 0,C 180,E1 -413.957,E2 -413.957} C_VEL
LIN {X 0,Y 608.53,Z 319.978,A -85,B 0,C 180,E1 -414.577,E2 -414.577} C_VEL
LIN {X 0,Y 608.526,Z 333.73,A -85,B 0,C 180,E1 -417.126,E2 -417.126} C_VEL
LIN {X 0,Y 608.588,Z 344.409,A -85,B 0,C 180,E1 -419.085,E2 -419.085} C_VEL
LIN {X 0,Y 608.589,Z 356.086,A -85,B 0,C 180,E1 -421.361,E2 -421.361} C_VEL
LIN {X 0,Y 608.572,Z 371.341,A -85,B 0,C 180,E1 -424.26,E2 -424.26} C_VEL
LIN {X 0,Y 608.52,Z 385.454,A -85,B 0,C 180,E1 -426.879,E2 -426.879} C_VEL
LIN {X 0,Y 608.478,Z 399.974,A -85,B 0,C 180,E1 -429.523,E2 -429.523} C_VEL
LIN {X 0,Y 608.483,Z 414.799,A -85,B 0,C 180,E1 -432.178,E2 -432.178} C_VEL
LIN {X 0,Y 608.451,Z 430.45,A -85,B 0,C 180,E1 -434.937,E2 -434.937} C_VEL
LIN {X 0,Y 608.435,Z 444.145,A -85,B 0,C 180,E1 -437.323,E2 -437.323} C_VEL
LIN {X 0,Y 608.463,Z 449.059,A -85,B 0,C 180,E1 -438.149,E2 -438.149} C_VEL
LIN {X 0,Y 608.539,Z 450.803,A -85,B 0,C 180,E1 -438.213,E2 -438.213} C_VEL
LIN {X 0,Y 608.523,Z 464.163,A -85,B 0,C 180,E1 -438.466,E2 -438.466} C_VEL
LIN {X 0,Y 608.516,Z 477.328,A -85,B 0,C 180,E1 -438.858,E2 -438.858} C_VEL
LIN {X 0,Y 608.517,Z 489.201,A -85,B 0,C 180,E1 -439.351,E2 -439.351} C_VEL
LIN {X 0,Y 608.491,Z 501.56,A -85,B 0,C 180,E1 -440.024,E2 -440.024} C_VEL
LIN {X 0,Y 608.483,Z 512.495,A -85,B 0,C 180,E1 -440.778,E2 -440.778} C_VEL
LIN {X 0,Y 608.459,Z 523.102,A -85,B 0,C 180,E1 -441.699,E2 -441.699} C_VEL
LIN {X 0,Y 608.47,Z 530.952,A -85,B 0,C 180,E1 -442.534,E2 -442.534} C_VEL
LIN {X 0,Y 608.461,Z 538.297,A -85,B 0,C 180,E1 -443.484,E2 -443.484} C_VEL
LIN {X 0,Y 608.451,Z 543.869,A -85,B 0,C 180,E1 -444.366,E2 -444.366} C_VEL
LIN {X 0,Y 608.431,Z 548.956,A -85,B 0,C 180,E1 -445.362,E2 -445.362} C_VEL
LIN {X 0,Y 608.449,Z 552.898,A -85,B 0,C 180,E1 -446.358,E2 -446.358} C_VEL
LIN {X 0,Y 608.425,Z 555.806,A -85,B 0,C 180,E1 -447.352,E2 -447.352} C_VEL
LIN {X 0,Y 608.444,Z 557.204,A -85,B 0,C 180,E1 -448.014,E2 -448.014} C_VEL
LIN {X 0,Y 608.439,Z 558.783,A -85,B 0,C 180,E1 -449.338,E2 -449.338} C_VEL
LIN {X 0,Y 608.434,Z 559,A -85,B 0,C 180,E1 -450,E2 -450} C_VEL
LIN {X 0,Y 608.448,Z 558.184,A -85,B 0,C 180,E1 -451.324,E2 -451.324} C_VEL
LIN {X 0,Y 608.444,Z 557.204,A -85,B 0,C 180,E1 -451.986,E2 -451.986} C_VEL
LIN {X 0,Y 608.425,Z 555.807,A -85,B 0,C 180,E1 -452.648,E2 -452.648} C_VEL
LIN {X 0,Y 608.449,Z 552.898,A -85,B 0,C 180,E1 -453.642,E2 -453.642} C_VEL
LIN {X 0,Y 608.431,Z 548.956,A -85,B 0,C 180,E1 -454.638,E2 -454.638} C_VEL
LIN {X 0,Y 608.451,Z 543.869,A -85,B 0,C 180,E1 -455.634,E2 -455.634} C_VEL
LIN {X 0,Y 608.443,Z 537.462,A -85,B 0,C 180,E1 -456.633,E2 -456.633} C_VEL
LIN {X 0,Y 608.475,Z 529.479,A -85,B 0,C 180,E1 -457.633,E2 -457.633} C_VEL
LIN {X 0,Y 608.487,Z 521.347,A -85,B 0,C 180,E1 -458.468,E2 -458.468} C_VEL
LIN {X 0,Y 608.487,Z 511.39,A -85,B 0,C 180,E1 -459.305,E2 -459.305} C_VEL
LIN {X 0,Y 608.516,Z 500.173,A -85,B 0,C 180,E1 -460.06,E2 -460.06} C_VEL
LIN {X 0,Y 608.517,Z 489.202,A -85,B 0,C 180,E1 -460.649,E2 -460.649} C_VEL
LIN {X 0,Y 608.521,Z 477.794,A -85,B 0,C 180,E1 -461.126,E2 -461.126} C_VEL
LIN {X 0,Y 608.511,Z 465.036,A -85,B 0,C 180,E1 -461.513,E2 -461.513} C_VEL
LIN {X 0,Y 608.53,Z 452.142,A -85,B 0,C 180,E1 -461.766,E2 -461.766} C_VEL
LIN {X 0,Y 608.486,Z 449.332,A -85,B 0,C 180,E1 -461.83,E2 -461.83} C_VEL
LIN {X 0,Y 608.435,Z 446.101,A -85,B 0,C 180,E1 -462.339,E2 -462.339} C_VEL
LIN {X 0,Y 608.452,Z 430.45,A -85,B 0,C 180,E1 -465.063,E2 -465.063} C_VEL
LIN {X 0,Y 608.483,Z 414.799,A -85,B 0,C 180,E1 -467.822,E2 -467.822} C_VEL
LIN {X 0,Y 608.48,Z 398.844,A -85,B 0,C 180,E1 -470.681,E2 -470.681} C_VEL
LIN {X 0,Y 608.52,Z 385.454,A -85,B 0,C 180,E1 -473.121,E2 -473.121} C_VEL
LIN {X 0,Y 608.567,Z 369.803,A -85,B 0,C 180,E1 -476.029,E2 -476.029} C_VEL
LIN {X 0,Y 608.589,Z 356.086,A -85,B 0,C 180,E1 -478.639,E2 -478.639} C_VEL
LIN {X 0,Y 608.609,Z 342.396,A -85,B 0,C 180,E1 -481.307,E2 -481.307} C_VEL
LIN {X 0,Y 608.616,Z 326.829,A -85,B 0,C 180,E1 -484.259,E2 -484.259} C_VEL
LIN {X 0,Y 608.518,Z 319.899,A -85,B 0,C 180,E1 -485.627,E2 -485.627} C_VEL
LIN {X 0,Y 608.404,Z 319.695,A -85,B 0,C 180,E1 -488.232,E2 -488.232} C_VEL
LIN {X 0,Y 608.427,Z 319.691,A -85,B 0,C 180,E1 -490.326,E2 -490.326} C_VEL
LIN {X 0,Y 608.429,Z 319.693,A -85,B 0,C 180,E1 -492.961,E2 -492.961} C_VEL
LIN {X 0,Y 608.429,Z 319.696,A -85,B 0,C 180,E1 -495.737,E2 -495.737} C_VEL
LIN {X 0,Y 608.43,Z 319.692,A -85,B 0,C 180,E1 -497.936,E2 -497.936} C_VEL
LIN {X 0,Y 608.422,Z 319.692,A -85,B 0,C 180,E1 -500.706,E2 -500.706} C_VEL
LIN {X 0,Y 608.452,Z 319.694,A -85,B 0,C 180,E1 -503.085,E2 -503.085} C_VEL
LIN {X 0,Y 608.463,Z 319.692,A -85,B 0,C 180,E1 -505.53,E2 -505.53} C_VEL
LIN {X 0,Y 608.436,Z 319.691,A -85,B 0,C 180,E1 -507.904,E2 -507.904} C_VEL
LIN {X 0,Y 608.423,Z 319.691,A -85,B 0,C 180,E1 -510.218,E2 -510.218} C_VEL
LIN {X 0,Y 608.477,Z 319.688,A -85,B 0,C 180,E1 -512.79,E2 -512.79} C_VEL
LIN {X 0,Y 608.442,Z 319.69,A -85,B 0,C 180,E1 -515.852,E2 -515.852} C_VEL
LIN {X 0,Y 608.438,Z 319.69,A -85,B 0,C 180,E1 -518.307,E2 -518.307} C_VEL
LIN {X 0,Y 608.46,Z 319.693,A -85,B 0,C 180,E1 -521.283,E2 -521.283} C_VEL
LIN {X 0,Y 608.426,Z 319.691,A -85,B 0,C 180,E1 -523.905,E2 -523.905} C_VEL
LIN {X 0,Y 608.462,Z 319.691,A -85,B 0,C 180,E1 -526.643,E2 -526.643} C_VEL
LIN {X 0,Y 608.449,Z 319.692,A -85,B 0,C 180,E1 -529.35,E2 -529.35} C_VEL
LIN {X 0,Y 608.435,Z 319.693,A -85,B 0,C 180,E1 -531.364,E2 -531.364} C_VEL
LIN {X 0,Y 608.444,Z 319.691,A -85,B 0,C 180,E1 -533.385,E2 -533.385} C_VEL
LIN {X 0,Y 608.422,Z 319.691,A -85,B 0,C 180,E1 -536.026,E2 -536.026} C_VEL
LIN {X 0,Y 608.476,Z 319.693,A -85,B 0,C 180,E1 -538.676,E2 -538.676} C_VEL
LIN {X 0,Y 608.45,Z 319.69,A -85,B 0,C 180,E1 -541.324,E2 -541.324} C_VEL
LIN {X 0,Y 608.46,Z 319.689,A -85,B 0,C 180,E1 -543.311,E2 -543.311} C_VEL
LIN {X 0,Y 608.435,Z 319.69,A -85,B 0,C 180,E1 -545.967,E2 -545.967} C_VEL
LIN {X 0,Y 608.457,Z 319.697,A -85,B 0,C 180,E1 -548.636,E2 -548.636} C_VEL
LIN {X 0,Y 608.439,Z 319.689,A -85,B 0,C 180,E1 -549.476,E2 -549.476} C_VEL
LIN {X 0,Y 607.759,Z 319.776,A -85,B 0,C 180,E1 -550.029,E2 -550.029} C_VEL
LIN {X 0,Y 604.904,Z 320.135,A -85,B 0,C 180,E1 -550.926,E2 -550.926} C_VEL
LIN {X 0,Y 602.504,Z 320.432,A -85,B 0,C 180,E1 -551.648,E2 -551.648} C_VEL
LIN {X 0,Y 601.48,Z 320.559,A -85,B 0,C 180,E1 -552.205,E2 -552.205} C_VEL
LIN {X 0,Y 601.4,Z 320.569,A -85,B 0,C 180,E1 -552.393,E2 -552.393} C_VEL
LIN {X 0,Y 601.421,Z 320.569,A -85,B 0,C 180,E1 -554.897,E2 -554.897} C_VEL
LIN {X 0,Y 601.422,Z 320.567,A -85,B 0,C 180,E1 -556.986,E2 -556.986} C_VEL
LIN {X 0,Y 601.396,Z 320.567,A -85,B 0,C 180,E1 -559.81,E2 -559.81} C_VEL
LIN {X 0,Y 601.446,Z 320.567,A -85,B 0,C 180,E1 -562.682,E2 -562.682} C_VEL
LIN {X 0,Y 601.392,Z 320.571,A -85,B 0,C 180,E1 -564.879,E2 -564.879} C_VEL
LIN {X 0,Y 601.416,Z 320.566,A -85,B 0,C 180,E1 -567.868,E2 -567.868} C_VEL
LIN {X 0,Y 601.44,Z 320.568,A -85,B 0,C 180,E1 -570.163,E2 -570.163} C_VEL
LIN {X 0,Y 601.422,Z 320.567,A -85,B 0,C 180,E1 -572.718,E2 -572.718} C_VEL
LIN {X 0,Y 601.387,Z 320.568,A -85,B 0,C 180,E1 -575.113,E2 -575.113} C_VEL
LIN {X 0,Y 601.426,Z 320.563,A -85,B 0,C 180,E1 -577.42,E2 -577.42} C_VEL
LIN {X 0,Y 601.403,Z 320.572,A -85,B 0,C 180,E1 -579.996,E2 -579.996} C_VEL
LIN {X 0,Y 601.406,Z 320.568,A -85,B 0,C 180,E1 -582.671,E2 -582.671} C_VEL
LIN {X 0,Y 601.421,Z 320.564,A -85,B 0,C 180,E1 -585.483,E2 -585.483} C_VEL
LIN {X 0,Y 601.422,Z 320.569,A -85,B 0,C 180,E1 -588.407,E2 -588.407} C_VEL
LIN {X 0,Y 601.429,Z 320.564,A -85,B 0,C 180,E1 -591.53,E2 -591.53} C_VEL
LIN {X 0,Y 601.407,Z 320.572,A -85,B 0,C 180,E1 -594.248,E2 -594.248} C_VEL
LIN {X 0,Y 601.428,Z 320.564,A -85,B 0,C 180,E1 -596.687,E2 -596.687} C_VEL
LIN {X 0,Y 601.448,Z 320.568,A -85,B 0,C 180,E1 -599.838,E2 -599.838} C_VEL
LIN {X 0,Y 601.41,Z 320.566,A -85,B 0,C 180,E1 -602.639,E2 -602.639} C_VEL
LIN {X 0,Y 601.4,Z 320.566,A -85,B 0,C 180,E1 -605.122,E2 -605.122} C_VEL
LIN {X 0,Y 601.416,Z 320.567,A -85,B 0,C 180,E1 -607.395,E2 -607.395} C_VEL
LIN {X 0,Y 601.407,Z 320.569,A -85,B 0,C 180,E1 -610.191,E2 -610.191} C_VEL
LIN {X 0,Y 601.433,Z 320.562,A -85,B 0,C 180,E1 -613.015,E2 -613.015} C_VEL
LIN {X 0,Y 601.425,Z 320.57,A -85,B 0,C 180,E1 -615.908,E2 -615.908} C_VEL
LIN {X 0,Y 601.416,Z 320.564,A -85,B 0,C 180,E1 -618.542,E2 -618.542} C_VEL
LIN {X 0,Y 601.44,Z 320.565,A -85,B 0,C 180,E1 -621.263,E2 -621.263} C_VEL
LIN {X 0,Y 601.442,Z 320.565,A -85,B 0,C 180,E1 -623.963,E2 -623.963} C_VEL
LIN {X 0,Y 601.426,Z 320.563,A -85,B 0,C 180,E1 -626.651,E2 -626.651} C_VEL
LIN {X 0,Y 601.458,Z 320.565,A -85,B 0,C 180,E1 -629.331,E2 -629.331} C_VEL
LIN {X 0,Y 601.437,Z 320.564,A -85,B 0,C 180,E1 -632.009,E2 -632.009} C_VEL
LIN {X 0,Y 601.418,Z 320.564,A -85,B 0,C 180,E1 -634.692,E2 -634.692} C_VEL
LIN {X 0,Y 601.447,Z 320.57,A -85,B 0,C 180,E1 -637.385,E2 -637.385} C_VEL
LIN {X 0,Y 601.439,Z 320.562,A -85,B 0,C 180,E1 -640.095,E2 -640.095} C_VEL
LIN {X 0,Y 601.423,Z 320.565,A -85,B 0,C 180,E1 -642.828,E2 -642.828} C_VEL
LIN {X 0,Y 601.417,Z 320.57,A -85,B 0,C 180,E1 -645.591,E2 -645.591} C_VEL
LIN {X 0,Y 601.425,Z 320.563,A -85,B 0,C 180,E1 -648.391,E2 -648.391} C_VEL
LIN {X 0,Y 601.412,Z 320.575,A -85,B 0,C 180,E1 -651.239,E2 -651.239} C_VEL
LIN {X 0,Y 601.456,Z 320.559,A -85,B 0,C 180,E1 -654.14,E2 -654.14} C_VEL
LIN {X 0,Y 601.457,Z 320.569,A -85,B 0,C 180,E1 -657.11,E2 -657.11} C_VEL
LIN {X 0,Y 601.425,Z 320.569,A -85,B 0,C 180,E1 -659.392,E2 -659.392} C_VEL
LIN {X 0,Y 601.416,Z 320.565,A -85,B 0,C 180,E1 -661.725,E2 -661.725} C_VEL
LIN {X 0,Y 601.43,Z 320.562,A -85,B 0,C 180,E1 -664.117,E2 -664.117} C_VEL
LIN {X 0,Y 601.417,Z 320.567,A -85,B 0,C 180,E1 -666.581,E2 -666.581} C_VEL
LIN {X 0,Y 601.441,Z 320.563,A -85,B 0,C 180,E1 -669.536,E2 -669.536} C_VEL
LIN {X 0,Y 601.438,Z 320.566,A -85,B 0,C 180,E1 -672.593,E2 -672.593} C_VEL
LIN {X 0,Y 601.42,Z 320.566,A -85,B 0,C 180,E1 -675.481,E2 -675.481} C_VEL
LIN {X 0,Y 601.425,Z 320.567,A -85,B 0,C 180,E1 -678.405,E2 -678.405} C_VEL
LIN {X 0,Y 601.429,Z 320.566,A -85,B 0,C 180,E1 -680.543,E2 -680.543} C_VEL
LIN {X 0,Y 601.555,Z 332.354,A -85,B 0,C 180,E1 -680.972,E2 -680.972} C_VEL
LIN {X 0,Y 601.515,Z 342.849,A -85,B 0,C 180,E1 -681.46,E2 -681.46} C_VEL
LIN {X 0,Y 601.477,Z 351.441,A -85,B 0,C 180,E1 -681.949,E2 -681.949} C_VEL
LIN {X 0,Y 601.458,Z 361.079,A -85,B 0,C 180,E1 -682.613,E2 -682.613} C_VEL
LIN {X 0,Y 601.424,Z 370.711,A -85,B 0,C 180,E1 -683.418,E2 -683.418} C_VEL
LIN {X 0,Y 601.394,Z 380.303,A -85,B 0,C 180,E1 -684.42,E2 -684.42} C_VEL
LIN {X 0,Y 601.377,Z 386.944,A -85,B 0,C 180,E1 -685.269,E2 -685.269} C_VEL
LIN {X 0,Y 601.373,Z 392.211,A -85,B 0,C 180,E1 -686.071,E2 -686.071} C_VEL
LIN {X 0,Y 601.343,Z 397.304,A -85,B 0,C 180,E1 -687.014,E2 -687.014} C_VEL
LIN {X 0,Y 601.334,Z 401.077,A -85,B 0,C 180,E1 -687.875,E2 -687.875} C_VEL
LIN {X 0,Y 601.343,Z 403.539,A -85,B 0,C 180,E1 -688.555,E2 -688.555} C_VEL
LIN {X 0,Y 601.334,Z 406.834,A -85,B 0,C 180,E1 -689.865,E2 -689.865} C_VEL
LIN {X 0,Y 601.33,Z 408.069,A -85,B 0,C 180,E1 -690.602,E2 -690.602} C_VEL
LIN {X 0,Y 601.329,Z 408.777,A -85,B 0,C 180,E1 -691.368,E2 -691.368} C_VEL
LIN {X 0,Y 601.343,Z 408.805,A -85,B 0,C 180,E1 -692.648,E2 -692.648} C_VEL
LIN {X 0,Y 601.308,Z 407.848,A -85,B 0,C 180,E1 -693.632,E2 -693.632} C_VEL
LIN {X 0,Y 601.324,Z 406.582,A -85,B 0,C 180,E1 -694.378,E2 -694.378} C_VEL
LIN {X 0,Y 601.347,Z 404.732,A -85,B 0,C 180,E1 -695.119,E2 -695.119} C_VEL
LIN {X 0,Y 601.353,Z 401.089,A -85,B 0,C 180,E1 -696.222,E2 -696.222} C_VEL
LIN {X 0,Y 601.37,Z 395.697,A -85,B 0,C 180,E1 -697.402,E2 -697.402} C_VEL
LIN {X 0,Y 601.392,Z 389.808,A -85,B 0,C 180,E1 -698.4,E2 -698.4} C_VEL
LIN {X 0,Y 601.409,Z 383.478,A -85,B 0,C 180,E1 -699.28,E2 -699.28} C_VEL
LIN {X 0,Y 601.424,Z 377.219,A -85,B 0,C 180,E1 -700.013,E2 -700.013} C_VEL
LIN {X 0,Y 601.421,Z 370.092,A -85,B 0,C 180,E1 -700.724,E2 -700.724} C_VEL
LIN {X 0,Y 601.471,Z 362.35,A -85,B 0,C 180,E1 -701.379,E2 -701.379} C_VEL
LIN {X 0,Y 601.493,Z 352.858,A -85,B 0,C 180,E1 -702.051,E2 -702.051} C_VEL
LIN {X 0,Y 601.521,Z 342.203,A -85,B 0,C 180,E1 -702.666,E2 -702.666} C_VEL
LIN {X 0,Y 601.554,Z 329.403,A -85,B 0,C 180,E1 -703.241,E2 -703.241} C_VEL
LIN {X 0,Y 601.575,Z 321.443,A -85,B 0,C 180,E1 -703.527,E2 -703.527} C_VEL
LIN {X 0,Y 601.458,Z 320.647,A -85,B 0,C 180,E1 -703.65,E2 -703.65} C_VEL
LIN {X 0,Y 601.4,Z 320.566,A -85,B 0,C 180,E1 -706.484,E2 -706.484} C_VEL
LIN {X 0,Y 601.421,Z 320.571,A -85,B 0,C 180,E1 -709.224,E2 -709.224} C_VEL
LIN {X 0,Y 601.424,Z 320.565,A -85,B 0,C 180,E1 -711.939,E2 -711.939} C_VEL
LIN {X 0,Y 601.41,Z 320.566,A -85,B 0,C 180,E1 -714.636,E2 -714.636} C_VEL
LIN {X 0,Y 601.446,Z 320.571,A -85,B 0,C 180,E1 -717.321,E2 -717.321} C_VEL
LIN {X 0,Y 601.417,Z 320.565,A -85,B 0,C 180,E1 -720,E2 -720} C_VEL
LIN {X 0,Y 601.424,Z 320.565,A -85,B 0,C 180,E1 -722.679,E2 -722.679} C_VEL
LIN {X 0,Y 601.428,Z 320.571,A -85,B 0,C 180,E1 -725.364,E2 -725.364} C_VEL
LIN {X 0,Y 601.393,Z 320.567,A -85,B 0,C 180,E1 -728.061,E2 -728.061} C_VEL
LIN {X 0,Y 601.408,Z 320.569,A -85,B 0,C 180,E1 -730.776,E2 -730.776} C_VEL
LIN {X 0,Y 601.403,Z 320.57,A -85,B 0,C 180,E1 -733.516,E2 -733.516} C_VEL
LIN {X 0,Y 601.411,Z 320.565,A -85,B 0,C 180,E1 -736.288,E2 -736.288} C_VEL
LIN {X 0,Y 601.405,Z 320.575,A -85,B 0,C 180,E1 -739.099,E2 -739.099} C_VEL
LIN {X 0,Y 601.392,Z 320.574,A -85,B 0,C 180,E1 -741.24,E2 -741.24} C_VEL
LIN {X 0,Y 601.421,Z 320.563,A -85,B 0,C 180,E1 -744.142,E2 -744.142} C_VEL
LIN {X 0,Y 601.448,Z 320.568,A -85,B 0,C 180,E1 -747.111,E2 -747.111} C_VEL
LIN {X 0,Y 601.391,Z 320.57,A -85,B 0,C 180,E1 -749.395,E2 -749.395} C_VEL
LIN {X 0,Y 601.381,Z 320.569,A -85,B 0,C 180,E1 -751.728,E2 -751.728} C_VEL
LIN {X 0,Y 601.404,Z 320.566,A -85,B 0,C 180,E1 -754.12,E2 -754.12} C_VEL
LIN {X 0,Y 601.422,Z 320.565,A -85,B 0,C 180,E1 -757.382,E2 -757.382} C_VEL
LIN {X 0,Y 601.388,Z 320.568,A -85,B 0,C 180,E1 -759.997,E2 -759.997} C_VEL
LIN {X 0,Y 601.399,Z 320.576,A -85,B 0,C 180,E1 -762.672,E2 -762.672} C_VEL
LIN {X 0,Y 601.392,Z 320.568,A -85,B 0,C 180,E1 -765.48,E2 -765.48} C_VEL
LIN {X 0,Y 601.413,Z 320.571,A -85,B 0,C 180,E1 -768.408,E2 -768.408} C_VEL
LIN {X 0,Y 601.388,Z 320.575,A -85,B 0,C 180,E1 -770.873,E2 -770.873} C_VEL
LIN {X 0,Y 601.376,Z 320.572,A -85,B 0,C 180,E1 -773.416,E2 -773.416} C_VEL
LIN {X 0,Y 601.449,Z 320.72,A -85,B 0,C 180,E1 -774.378,E2 -774.378} C_VEL
LIN {X 0,Y 601.608,Z 325.353,A -85,B 0,C 180,E1 -775.286,E2 -775.286} C_VEL
LIN {X 0,Y 601.621,Z 341.568,A -85,B 0,C 180,E1 -778.287,E2 -778.287} C_VEL
LIN {X 0,Y 601.726,Z 352.196,A -85,B 0,C 180,E1 -780.239,E2 -780.239} C_VEL
LIN {X 0,Y 601.626,Z 365.89,A -85,B 0,C 180,E1 -782.898,E2 -782.898} C_VEL
LIN {X 0,Y 601.592,Z 379.345,A -85,B 0,C 180,E1 -785.454,E2 -785.454} C_VEL
LIN {X 0,Y 601.549,Z 393.279,A -85,B 0,C 180,E1 -788.047,E2 -788.047} C_VEL
LIN {X 0,Y 601.476,Z 408.93,A -85,B 0,C 180,E1 -790.903,E2 -790.903} C_VEL
LIN {X 0,Y 601.433,Z 422.696,A -85,B 0,C 180,E1 -793.377,E2 -793.377} C_VEL
LIN {X 0,Y 601.434,Z 438.599,A -85,B 0,C 180,E1 -796.197,E2 -796.197} C_VEL
LIN {X 0,Y 601.426,Z 449.057,A -85,B 0,C 180,E1 -798.008,E2 -798.008} C_VEL
LIN {X 0,Y 601.583,Z 450.783,A -85,B 0,C 180,E1 -798.075,E2 -798.075} C_VEL
LIN {X 0,Y 601.574,Z 464.163,A -85,B 0,C 180,E1 -798.331,E2 -798.331} C_VEL
LIN {X 0,Y 601.549,Z 477.202,A -85,B 0,C 180,E1 -798.722,E2 -798.722} C_VEL
LIN {X 0,Y 601.525,Z 489.202,A -85,B 0,C 180,E1 -799.226,E2 -799.226} C_VEL
LIN {X 0,Y 601.491,Z 501.561,A -85,B 0,C 180,E1 -799.906,E2 -799.906} C_VEL
LIN {X 0,Y 601.449,Z 512.495,A -85,B 0,C 180,E1 -800.67,E2 -800.67} C_VEL
LIN {X 0,Y 601.405,Z 523.101,A -85,B 0,C 180,E1 -801.601,E2 -801.601} C_VEL
LIN {X 0,Y 601.417,Z 530.951,A -85,B 0,C 180,E1 -802.446,E2 -802.446} C_VEL
LIN {X 0,Y 601.37,Z 538.235,A -85,B 0,C 180,E1 -803.398,E2 -803.398} C_VEL
LIN {X 0,Y 601.374,Z 543.869,A -85,B 0,C 180,E1 -804.299,E2 -804.299} C_VEL
LIN {X 0,Y 601.335,Z 548.956,A -85,B 0,C 180,E1 -805.307,E2 -805.307} C_VEL
LIN {X 0,Y 601.367,Z 552.898,A -85,B 0,C 180,E1 -806.315,E2 -806.315} C_VEL
LIN {X 0,Y 601.324,Z 555.806,A -85,B 0,C 180,E1 -807.321,E2 -807.321} C_VEL
LIN {X 0,Y 601.343,Z 557.204,A -85,B 0,C 180,E1 -807.991,E2 -807.991} C_VEL
LIN {X 0,Y 601.339,Z 558.783,A -85,B 0,C 180,E1 -809.33,E2 -809.33} C_VEL
LIN {X 0,Y 601.335,Z 559,A -85,B 0,C 180,E1 -810,E2 -810} C_VEL
LIN {X 0,Y 601.347,Z 558.185,A -85,B 0,C 180,E1 -811.339,E2 -811.339} C_VEL
LIN {X 0,Y 601.343,Z 557.204,A -85,B 0,C 180,E1 -812.009,E2 -812.009} C_VEL
LIN {X 0,Y 601.324,Z 555.807,A -85,B 0,C 180,E1 -812.679,E2 -812.679} C_VEL
LIN {X 0,Y 601.367,Z 552.898,A -85,B 0,C 180,E1 -813.685,E2 -813.685} C_VEL
LIN {X 0,Y 601.335,Z 548.955,A -85,B 0,C 180,E1 -814.693,E2 -814.693} C_VEL
LIN {X 0,Y 601.374,Z 543.869,A -85,B 0,C 180,E1 -815.701,E2 -815.701} C_VEL
LIN {X 0,Y 601.382,Z 537.462,A -85,B 0,C 180,E1 -816.711,E2 -816.711} C_VEL
LIN {X 0,Y 601.396,Z 529.479,A -85,B 0,C 180,E1 -817.723,E2 -817.723} C_VEL
LIN {X 0,Y 601.423,Z 521.347,A -85,B 0,C 180,E1 -818.568,E2 -818.568} C_VEL
LIN {X 0,Y 601.455,Z 511.391,A -85,B 0,C 180,E1 -819.415,E2 -819.415} C_VEL
LIN {X 0,Y 601.507,Z 500.174,A -85,B 0,C 180,E1 -820.179,E2 -820.179} C_VEL
LIN {X 0,Y 601.525,Z 489.203,A -85,B 0,C 180,E1 -820.774,E2 -820.774} C_VEL
LIN {X 0,Y 601.562,Z 477.632,A -85,B 0,C 180,E1 -821.262,E2 -821.262} C_VEL
LIN {X 0,Y 601.578,Z 465.036,A -85,B 0,C 180,E1 -821.647,E2 -821.647} C_VEL
LIN {X 0,Y 601.604,Z 452.143,A -85,B 0,C 180,E1 -821.903,E2 -821.903} C_VEL
LIN {X 0,Y 601.455,Z 449.325,A -85,B 0,C 180,E1 -821.97,E2 -821.97} C_VEL
LIN {X 0,Y 601.378,Z 444.145,A -85,B 0,C 180,E1 -822.829,E2 -822.829} C_VEL
LIN {X 0,Y 601.447,Z 428.494,A -85,B 0,C 180,E1 -825.59,E2 -825.59} C_VEL
LIN {X 0,Y 601.477,Z 412.843,A -85,B 0,C 180,E1 -828.39,E2 -828.39} C_VEL
LIN {X 0,Y 601.526,Z 397.192,A -85,B 0,C 180,E1 -831.234,E2 -831.234} C_VEL
LIN {X 0,Y 601.591,Z 383.498,A -85,B 0,C 180,E1 -833.768,E2 -833.768} C_VEL
LIN {X 0,Y 601.628,Z 369.803,A -85,B 0,C 180,E1 -836.352,E2 -836.352} C_VEL
LIN {X 0,Y 601.712,Z 355.794,A -85,B 0,C 180,E1 -839.055,E2 -839.055} C_VEL
LIN {X 0,Y 601.678,Z 346.052,A -85,B 0,C 180,E1 -840.926,E2 -840.926} C_VEL
LIN {X 0,Y 601.698,Z 330.143,A -85,B 0,C 180,E1 -843.973,E2 -843.973} C_VEL
LIN {X 0,Y 601.735,Z 322.922,A -85,B 0,C 180,E1 -845.397,E2 -845.397} C_VEL
LIN {X 0,Y 601.435,Z 320.686,A -85,B 0,C 180,E1 -845.884,E2 -845.884} C_VEL
LIN {X 0,Y 601.373,Z 320.571,A -85,B 0,C 180,E1 -848.463,E2 -848.463} C_VEL
LIN {X 0,Y 601.402,Z 320.568,A -85,B 0,C 180,E1 -850.874,E2 -850.874} C_VEL
LIN {X 0,Y 601.422,Z 320.572,A -85,B 0,C 180,E1 -853.585,E2 -853.585} C_VEL
LIN {X 0,Y 601.395,Z 320.567,A -85,B 0,C 180,E1 -856.429,E2 -856.429} C_VEL
LIN {X 0,Y 601.398,Z 320.576,A -85,B 0,C 180,E1 -859.427,E2 -859.427} C_VEL
LIN {X 0,Y 601.391,Z 320.571,A -85,B 0,C 180,E1 -861.73,E2 -861.73} C_VEL
LIN {X 0,Y 601.368,Z 320.57,A -85,B 0,C 180,E1 -864.244,E2 -864.244} C_VEL
LIN {X 0,Y 601.404,Z 320.567,A -85,B 0,C 180,E1 -866.685,E2 -866.685} C_VEL
LIN {X 0,Y 601.394,Z 320.574,A -85,B 0,C 180,E1 -869.056,E2 -869.056} C_VEL
LIN {X 0,Y 601.425,Z 320.57,A -85,B 0,C 180,E1 -871.373,E2 -871.373} C_VEL
LIN {X 0,Y 601.386,Z 320.571,A -85,B 0,C 180,E1 -873.635,E2 -873.635} C_VEL
LIN {X 0,Y 601.421,Z 320.564,A -85,B 0,C 180,E1 -875.858,E2 -875.858} C_VEL
LIN {X 0,Y 601.392,Z 320.572,A -85,B 0,C 180,E1 -878.76,E2 -878.76} C_VEL
LIN {X 0,Y 601.382,Z 320.57,A -85,B 0,C 180,E1 -881.607,E2 -881.607} C_VEL
LIN {X 0,Y 601.411,Z 320.566,A -85,B 0,C 180,E1 -883.712,E2 -883.712} C_VEL
LIN {X 0,Y 601.403,Z 320.568,A -85,B 0,C 180,E1 -886.484,E2 -886.484} C_VEL
LIN {X 0,Y 601.407,Z 320.571,A -85,B 0,C 180,E1 -889.224,E2 -889.224} C_VEL
LIN {X 0,Y 601.393,Z 320.567,A -85,B 0,C 180,E1 -891.939,E2 -891.939} C_VEL
LIN {X 0,Y 601.428,Z 320.569,A -85,B 0,C 180,E1 -894.636,E2 -894.636} C_VEL
LIN {X 0,Y 601.424,Z 320.566,A -85,B 0,C 180,E1 -897.321,E2 -897.321} C_VEL
LIN {X 0,Y 601.417,Z 320.564,A -85,B 0,C 180,E1 -900,E2 -900} C_VEL
LIN {X 0,Y 601.446,Z 320.569,A -85,B 0,C 180,E1 -902.679,E2 -902.679} C_VEL
LIN {X 0,Y 601.41,Z 320.566,A -85,B 0,C 180,E1 -905.364,E2 -905.364} C_VEL
LIN {X 0,Y 601.423,Z 320.565,A -85,B 0,C 180,E1 -908.061,E2 -908.061} C_VEL
LIN {X 0,Y 601.424,Z 320.567,A -85,B 0,C 180,E1 -911.019,E2 -911.019} C_VEL
LIN {X 0,Y 601.4,Z 320.569,A -85,B 0,C 180,E1 -912.393,E2 -912.393} C_VEL
LIN {X 0,Y 600.741,Z 320.655,A -85,B 0,C 180,E1 -912.953,E2 -912.953} C_VEL
LIN {X 0,Y 597.89,Z 321.009,A -85,B 0,C 180,E1 -913.86,E2 -913.86} C_VEL
LIN {X 0,Y 595.475,Z 321.315,A -85,B 0,C 180,E1 -914.591,E2 -914.591} C_VEL
LIN {X 0,Y 594.434,Z 321.436,A -85,B 0,C 180,E1 -915.154,E2 -915.154} C_VEL
LIN {X 0,Y 594.348,Z 321.445,A -85,B 0,C 180,E1 -915.345,E2 -915.345} C_VEL
LIN {X 0,Y 594.378,Z 321.442,A -85,B 0,C 180,E1 -917.194,E2 -917.194} C_VEL
LIN {X 0,Y 594.369,Z 321.445,A -85,B 0,C 180,E1 -920.054,E2 -920.054} C_VEL
LIN {X 0,Y 594.388,Z 321.442,A -85,B 0,C 180,E1 -922.966,E2 -922.966} C_VEL
LIN {X 0,Y 594.362,Z 321.443,A -85,B 0,C 180,E1 -925.194,E2 -925.194} C_VEL
LIN {X 0,Y 594.376,Z 321.441,A -85,B 0,C 180,E1 -927.527,E2 -927.527} C_VEL
LIN {X 0,Y 594.39,Z 321.449,A -85,B 0,C 180,E1 -930.331,E2 -930.331} C_VEL
LIN {X 0,Y 594.371,Z 321.443,A -85,B 0,C 180,E1 -932.951,E2 -932.951} C_VEL
LIN {X 0,Y 594.348,Z 321.444,A -85,B 0,C 180,E1 -935.409,E2 -935.409} C_VEL
LIN {X 0,Y 594.384,Z 321.445,A -85,B 0,C 180,E1 -937.941,E2 -937.941} C_VEL
LIN {X 0,Y 594.376,Z 321.443,A -85,B 0,C 180,E1 -940.823,E2 -940.823} C_VEL
LIN {X 0,Y 594.36,Z 321.443,A -85,B 0,C 180,E1 -943.3,E2 -943.3} C_VEL
LIN {X 0,Y 594.378,Z 321.451,A -85,B 0,C 180,E1 -946.16,E2 -946.16} C_VEL
LIN {X 0,Y 594.372,Z 321.441,A -85,B 0,C 180,E1 -949.179,E2 -949.179} C_VEL
LIN {X 0,Y 594.385,Z 321.45,A -85,B 0,C 180,E1 -952.06,E2 -952.06} C_VEL
LIN {X 0,Y 594.353,Z 321.445,A -85,B 0,C 180,E1 -954.677,E2 -954.677} C_VEL
LIN {X 0,Y 594.378,Z 321.441,A -85,B 0,C 180,E1 -957.089,E2 -957.089} C_VEL
LIN {X 0,Y 594.398,Z 321.444,A -85,B 0,C 180,E1 -959.67,E2 -959.67} C_VEL
LIN {X 0,Y 594.374,Z 321.443,A -85,B 0,C 180,E1 -962.54,E2 -962.54} C_VEL
LIN {X 0,Y 594.376,Z 321.441,A -85,B 0,C 180,E1 -964.808,E2 -964.808} C_VEL
LIN {X 0,Y 594.365,Z 321.444,A -85,B 0,C 180,E1 -967.265,E2 -967.265} C_VEL
LIN {X 0,Y 594.378,Z 321.449,A -85,B 0,C 180,E1 -969.947,E2 -969.947} C_VEL
LIN {X 0,Y 594.39,Z 321.439,A -85,B 0,C 180,E1 -972.807,E2 -972.807} C_VEL
LIN {X 0,Y 594.392,Z 321.448,A -85,B 0,C 180,E1 -975.826,E2 -975.826} C_VEL
LIN {X 0,Y 594.384,Z 321.441,A -85,B 0,C 180,E1 -978.404,E2 -978.404} C_VEL
LIN {X 0,Y 594.401,Z 321.44,A -85,B 0,C 180,E1 -981.158,E2 -981.158} C_VEL
LIN {X 0,Y 594.393,Z 321.445,A -85,B 0,C 180,E1 -983.891,E2 -983.891} C_VEL
LIN {X 0,Y 594.378,Z 321.441,A -85,B 0,C 180,E1 -986.611,E2 -986.611} C_VEL
LIN {X 0,Y 594.429,Z 321.441,A -85,B 0,C 180,E1 -989.323,E2 -989.323} C_VEL
LIN {X 0,Y 594.406,Z 321.44,A -85,B 0,C 180,E1 -992.033,E2 -992.033} C_VEL
LIN {X 0,Y 594.389,Z 321.44,A -85,B 0,C 180,E1 -994.748,E2 -994.748} C_VEL
LIN {X 0,Y 594.399,Z 321.448,A -85,B 0,C 180,E1 -997.473,E2 -997.473} C_VEL
LIN {X 0,Y 594.398,Z 321.438,A -85,B 0,C 180,E1 -1000.216,E2 -1000.216} C_VEL
LIN {X 0,Y 594.371,Z 321.446,A -85,B 0,C 180,E1 -1002.983,E2 -1002.983} C_VEL
LIN {X 0,Y 594.37,Z 321.445,A -85,B 0,C 180,E1 -1005.78,E2 -1005.78} C_VEL
LIN {X 0,Y 594.389,Z 321.44,A -85,B 0,C 180,E1 -1008.617,E2 -1008.617} C_VEL
LIN {X 0,Y 594.371,Z 321.447,A -85,B 0,C 180,E1 -1011.503,E2 -1011.503} C_VEL
LIN {X 0,Y 594.389,Z 321.44,A -85,B 0,C 180,E1 -1014.445,E2 -1014.445} C_VEL
LIN {X 0,Y 594.391,Z 321.442,A -85,B 0,C 180,E1 -1016.698,E2 -1016.698} C_VEL
LIN {X 0,Y 594.385,Z 321.448,A -85,B 0,C 180,E1 -1018.997,E2 -1018.997} C_VEL
LIN {X 0,Y 594.394,Z 321.441,A -85,B 0,C 180,E1 -1021.645,E2 -1021.645} C_VEL
LIN {X 0,Y 594.395,Z 321.441,A -85,B 0,C 180,E1 -1024.578,E2 -1024.578} C_VEL
LIN {X 0,Y 594.387,Z 321.449,A -85,B 0,C 180,E1 -1027.085,E2 -1027.085} C_VEL
LIN {X 0,Y 594.376,Z 321.442,A -85,B 0,C 180,E1 -1029.774,E2 -1029.774} C_VEL
LIN {X 0,Y 594.386,Z 321.442,A -85,B 0,C 180,E1 -1032.373,E2 -1032.373} C_VEL
LIN {X 0,Y 594.358,Z 321.449,A -85,B 0,C 180,E1 -1035.19,E2 -1035.19} C_VEL
LIN {X 0,Y 594.384,Z 321.442,A -85,B 0,C 180,E1 -1037.626,E2 -1037.626} C_VEL
LIN {X 0,Y 594.396,Z 321.453,A -85,B 0,C 180,E1 -1040.431,E2 -1040.431} C_VEL
LIN {X 0,Y 594.583,Z 333.367,A -85,B 0,C 180,E1 -1040.884,E2 -1040.884} C_VEL
LIN {X 0,Y 594.535,Z 343.04,A -85,B 0,C 180,E1 -1041.343,E2 -1041.343} C_VEL
LIN {X 0,Y 594.491,Z 353.493,A -85,B 0,C 180,E1 -1041.96,E2 -1041.96} C_VEL
LIN {X 0,Y 594.424,Z 363.992,A -85,B 0,C 180,E1 -1042.726,E2 -1042.726} C_VEL
LIN {X 0,Y 594.359,Z 373.968,A -85,B 0,C 180,E1 -1043.636,E2 -1043.636} C_VEL
LIN {X 0,Y 594.335,Z 380.744,A -85,B 0,C 180,E1 -1044.382,E2 -1044.382} C_VEL
LIN {X 0,Y 594.309,Z 387.239,A -85,B 0,C 180,E1 -1045.231,E2 -1045.231} C_VEL
LIN {X 0,Y 594.292,Z 393.54,A -85,B 0,C 180,E1 -1046.233,E2 -1046.233} C_VEL
LIN {X 0,Y 594.257,Z 397.998,A -85,B 0,C 180,E1 -1047.104,E2 -1047.104} C_VEL
LIN {X 0,Y 594.251,Z 401.157,A -85,B 0,C 180,E1 -1047.846,E2 -1047.846} C_VEL
LIN {X 0,Y 594.245,Z 404.991,A -85,B 0,C 180,E1 -1049.038,E2 -1049.038} C_VEL
LIN {X 0,Y 594.221,Z 407.502,A -85,B 0,C 180,E1 -1050.215,E2 -1050.215} C_VEL
LIN {X 0,Y 594.245,Z 408.521,A -85,B 0,C 180,E1 -1051.064,E2 -1051.064} C_VEL
LIN {X 0,Y 594.218,Z 408.923,A -85,B 0,C 180,E1 -1051.765,E2 -1051.765} C_VEL
LIN {X 0,Y 594.251,Z 408.882,A -85,B 0,C 180,E1 -1052.533,E2 -1052.533} C_VEL
LIN {X 0,Y 594.216,Z 408.314,A -85,B 0,C 180,E1 -1053.292,E2 -1053.292} C_VEL
LIN {X 0,Y 594.219,Z 407.206,A -85,B 0,C 180,E1 -1054.048,E2 -1054.048} C_VEL
LIN {X 0,Y 594.25,Z 404.691,A -85,B 0,C 180,E1 -1055.175,E2 -1055.175} C_VEL
LIN {X 0,Y 594.257,Z 401.016,A -85,B 0,C 180,E1 -1056.29,E2 -1056.29} C_VEL
LIN {X 0,Y 594.275,Z 395.388,A -85,B 0,C 180,E1 -1057.522,E2 -1057.522} C_VEL
LIN {X 0,Y 594.321,Z 389.691,A -85,B 0,C 180,E1 -1058.495,E2 -1058.495} C_VEL
LIN {X 0,Y 594.351,Z 383.192,A -85,B 0,C 180,E1 -1059.404,E2 -1059.404} C_VEL
LIN {X 0,Y 594.355,Z 375.391,A -85,B 0,C 180,E1 -1060.306,E2 -1060.306} C_VEL
LIN {X 0,Y 594.39,Z 366.556,A -85,B 0,C 180,E1 -1061.151,E2 -1061.151} C_VEL
LIN {X 0,Y 594.464,Z 355.327,A -85,B 0,C 180,E1 -1062.009,E2 -1062.009} C_VEL
LIN {X 0,Y 594.511,Z 345.159,A -85,B 0,C 180,E1 -1062.633,E2 -1062.633} C_VEL
LIN {X 0,Y 594.572,Z 334.74,A -85,B 0,C 180,E1 -1063.147,E2 -1063.147} C_VEL
LIN {X 0,Y 594.517,Z 322.135,A -85,B 0,C 180,E1 -1063.65,E2 -1063.65} C_VEL
LIN {X 0,Y 594.422,Z 321.487,A -85,B 0,C 180,E1 -1063.78,E2 -1063.78} C_VEL
LIN {X 0,Y 594.367,Z 321.443,A -85,B 0,C 180,E1 -1066.321,E2 -1066.321} C_VEL
LIN {X 0,Y 594.376,Z 321.446,A -85,B 0,C 180,E1 -1069.095,E2 -1069.095} C_VEL
LIN {X 0,Y 594.402,Z 321.441,A -85,B 0,C 180,E1 -1071.843,E2 -1071.843} C_VEL
LIN {X 0,Y 594.374,Z 321.442,A -85,B 0,C 180,E1 -1074.572,E2 -1074.572} C_VEL
LIN {X 0,Y 594.409,Z 321.447,A -85,B 0,C 180,E1 -1077.289,E2 -1077.289} C_VEL
LIN {X 0,Y 594.388,Z 321.441,A -85,B 0,C 180,E1 -1080,E2 -1080} C_VEL
LIN {X 0,Y 594.391,Z 321.441,A -85,B 0,C 180,E1 -1082.711,E2 -1082.711} C_VEL
LIN {X 0,Y 594.389,Z 321.446,A -85,B 0,C 180,E1 -1085.428,E2 -1085.428} C_VEL
LIN {X 0,Y 594.346,Z 321.445,A -85,B 0,C 180,E1 -1088.158,E2 -1088.158} C_VEL
LIN {X 0,Y 594.38,Z 321.45,A -85,B 0,C 180,E1 -1091.076,E2 -1091.076} C_VEL
LIN {X 0,Y 594.362,Z 321.445,A -85,B 0,C 180,E1 -1093.679,E2 -1093.679} C_VEL
LIN {X 0,Y 594.376,Z 321.446,A -85,B 0,C 180,E1 -1096.718,E2 -1096.718} C_VEL
LIN {X 0,Y 594.353,Z 321.449,A -85,B 0,C 180,E1 -1099.335,E2 -1099.335} C_VEL
LIN {X 0,Y 594.345,Z 321.448,A -85,B 0,C 180,E1 -1101.504,E2 -1101.504} C_VEL
LIN {X 0,Y 594.376,Z 321.443,A -85,B 0,C 180,E1 -1104.447,E2 -1104.447} C_VEL
LIN {X 0,Y 594.376,Z 321.443,A -85,B 0,C 180,E1 -1107.527,E2 -1107.527} C_VEL
LIN {X 0,Y 594.357,Z 321.446,A -85,B 0,C 180,E1 -1110.326,E2 -1110.326} C_VEL
LIN {X 0,Y 594.367,Z 321.451,A -85,B 0,C 180,E1 -1112.951,E2 -1112.951} C_VEL
LIN {X 0,Y 594.339,Z 321.448,A -85,B 0,C 180,E1 -1115.41,E2 -1115.41} C_VEL
LIN {X 0,Y 594.364,Z 321.443,A -85,B 0,C 180,E1 -1117.943,E2 -1117.943} C_VEL
LIN {X 0,Y 594.358,Z 321.453,A -85,B 0,C 180,E1 -1120.822,E2 -1120.822} C_VEL
LIN {X 0,Y 594.341,Z 321.448,A -85,B 0,C 180,E1 -1123.302,E2 -1123.302} C_VEL
LIN {X 0,Y 594.354,Z 321.447,A -85,B 0,C 180,E1 -1126.162,E2 -1126.162} C_VEL
LIN {X 0,Y 594.365,Z 321.446,A -85,B 0,C 180,E1 -1129.18,E2 -1129.18} C_VEL
LIN {X 0,Y 594.348,Z 321.448,A -85,B 0,C 180,E1 -1132.058,E2 -1132.058} C_VEL
LIN {X 0,Y 594.415,Z 321.669,A -85,B 0,C 180,E1 -1134.232,E2 -1134.232} C_VEL
LIN {X 0,Y 594.675,Z 325.688,A -85,B 0,C 180,E1 -1135.034,E2 -1135.034} C_VEL
LIN {X 0,Y 594.616,Z 340.734,A -85,B 0,C 180,E1 -1137.869,E2 -1137.869} C_VEL
LIN {X 0,Y 594.798,Z 355.971,A -85,B 0,C 180,E1 -1140.637,E2 -1140.637} C_VEL
LIN {X 0,Y 594.709,Z 369.803,A -85,B 0,C 180,E1 -1143.317,E2 -1143.317} C_VEL
LIN {X 0,Y 594.642,Z 383.498,A -85,B 0,C 180,E1 -1145.937,E2 -1145.937} C_VEL
LIN {X 0,Y 594.541,Z 398.921,A -85,B 0,C 180,E1 -1148.825,E2 -1148.825} C_VEL
LIN {X 0,Y 594.476,Z 414.799,A -85,B 0,C 180,E1 -1151.743,E2 -1151.743} C_VEL
LIN {X 0,Y 594.397,Z 430.45,A -85,B 0,C 180,E1 -1154.572,E2 -1154.572} C_VEL
LIN {X 0,Y 594.326,Z 444.145,A -85,B 0,C 180,E1 -1157.016,E2 -1157.016} C_VEL
LIN {X 0,Y 594.387,Z 449.326,A -85,B 0,C 180,E1 -1157.885,E2 -1157.885} C_VEL
LIN {X 0,Y 594.658,Z 453.547,A -85,B 0,C 180,E1 -1157.977,E2 -1157.977} C_VEL
LIN {X 0,Y 594.62,Z 466.762,A -85,B 0,C 180,E1 -1158.258,E2 -1158.258} C_VEL
LIN {X 0,Y 594.57,Z 478.63,A -85,B 0,C 180,E1 -1158.642,E2 -1158.642} C_VEL
LIN {X 0,Y 594.545,Z 490.917,A -85,B 0,C 180,E1 -1159.184,E2 -1159.184} C_VEL
LIN {X 0,Y 594.467,Z 502.939,A -85,B 0,C 180,E1 -1159.872,E2 -1159.872} C_VEL
LIN {X 0,Y 594.406,Z 513.544,A -85,B 0,C 180,E1 -1160.644,E2 -1160.644} C_VEL
LIN {X 0,Y 594.349,Z 523.101,A -85,B 0,C 180,E1 -1161.5,E2 -1161.5} C_VEL
LIN {X 0,Y 594.347,Z 530.951,A -85,B 0,C 180,E1 -1162.356,E2 -1162.356} C_VEL
LIN {X 0,Y 594.309,Z 538.677,A -85,B 0,C 180,E1 -1163.387,E2 -1163.387} C_VEL
LIN {X 0,Y 594.289,Z 545.677,A -85,B 0,C 180,E1 -1164.571,E2 -1164.571} C_VEL
LIN {X 0,Y 594.27,Z 550.368,A -85,B 0,C 180,E1 -1165.591,E2 -1165.591} C_VEL
LIN {X 0,Y 594.267,Z 553.955,A -85,B 0,C 180,E1 -1166.61,E2 -1166.61} C_VEL
LIN {X 0,Y 594.225,Z 555.807,A -85,B 0,C 180,E1 -1167.288,E2 -1167.288} C_VEL
LIN {X 0,Y 594.242,Z 557.203,A -85,B 0,C 180,E1 -1167.967,E2 -1167.967} C_VEL
LIN {X 0,Y 594.239,Z 558.784,A -85,B 0,C 180,E1 -1169.322,E2 -1169.322} C_VEL
LIN {X 0,Y 594.236,Z 559,A -85,B 0,C 180,E1 -1170,E2 -1170} C_VEL
LIN {X 0,Y 594.247,Z 558.185,A -85,B 0,C 180,E1 -1171.355,E2 -1171.355} C_VEL
LIN {X 0,Y 594.242,Z 557.204,A -85,B 0,C 180,E1 -1172.033,E2 -1172.033} C_VEL
LIN {X 0,Y 594.225,Z 555.807,A -85,B 0,C 180,E1 -1172.712,E2 -1172.712} C_VEL
LIN {X 0,Y 594.289,Z 552.898,A -85,B 0,C 180,E1 -1173.729,E2 -1173.729} C_VEL
LIN {X 0,Y 594.24,Z 548.955,A -85,B 0,C 180,E1 -1174.749,E2 -1174.749} C_VEL
LIN {X 0,Y 594.3,Z 543.869,A -85,B 0,C 180,E1 -1175.769,E2 -1175.769} C_VEL
LIN {X 0,Y 594.317,Z 537.462,A -85,B 0,C 180,E1 -1176.791,E2 -1176.791} C_VEL
LIN {X 0,Y 594.346,Z 529.48,A -85,B 0,C 180,E1 -1177.815,E2 -1177.815} C_VEL
LIN {X 0,Y 594.377,Z 521.347,A -85,B 0,C 180,E1 -1178.671,E2 -1178.671} C_VEL
LIN {X 0,Y 594.42,Z 511.392,A -85,B 0,C 180,E1 -1179.528,E2 -1179.528} C_VEL
LIN {X 0,Y 594.48,Z 500.175,A -85,B 0,C 180,E1 -1180.3,E2 -1180.3} C_VEL
LIN {X 0,Y 594.549,Z 489.202,A -85,B 0,C 180,E1 -1180.902,E2 -1180.902} C_VEL
LIN {X 0,Y 594.572,Z 476.838,A -85,B 0,C 180,E1 -1181.424,E2 -1181.424} C_VEL
LIN {X 0,Y 594.615,Z 463.287,A -85,B 0,C 180,E1 -1181.829,E2 -1181.829} C_VEL
LIN {X 0,Y 594.584,Z 450.763,A -85,B 0,C 180,E1 -1182.067,E2 -1182.067} C_VEL
LIN {X 0,Y 594.36,Z 449.047,A -85,B 0,C 180,E1 -1182.137,E2 -1182.137} C_VEL
LIN {X 0,Y 594.391,Z 434.363,A -85,B 0,C 180,E1 -1184.727,E2 -1184.727} C_VEL
LIN {X 0,Y 594.468,Z 418.712,A -85,B 0,C 180,E1 -1187.545,E2 -1187.545} C_VEL
LIN {X 0,Y 594.514,Z 403.061,A -85,B 0,C 180,E1 -1190.409,E2 -1190.409} C_VEL
LIN {X 0,Y 594.608,Z 389.367,A -85,B 0,C 180,E1 -1192.957,E2 -1192.957} C_VEL
LIN {X 0,Y 594.706,Z 373.716,A -85,B 0,C 180,E1 -1195.928,E2 -1195.928} C_VEL
LIN {X 0,Y 594.782,Z 360.021,A -85,B 0,C 180,E1 -1198.59,E2 -1198.59} C_VEL
LIN {X 0,Y 594.731,Z 346.547,A -85,B 0,C 180,E1 -1201.13,E2 -1201.13} C_VEL
LIN {X 0,Y 594.817,Z 330.779,A -85,B 0,C 180,E1 -1204.2,E2 -1204.2} C_VEL
LIN {X 0,Y 594.869,Z 324.848,A -85,B 0,C 180,E1 -1205.393,E2 -1205.393} C_VEL
LIN {X 0,Y 594.356,Z 321.527,A -85,B 0,C 180,E1 -1206.138,E2 -1206.138} C_VEL
LIN {X 0,Y 594.351,Z 321.447,A -85,B 0,C 180,E1 -1208.806,E2 -1208.806} C_VEL
LIN {X 0,Y 594.361,Z 321.448,A -85,B 0,C 180,E1 -1211.846,E2 -1211.846} C_VEL
LIN {X 0,Y 594.354,Z 321.445,A -85,B 0,C 180,E1 -1214.238,E2 -1214.238} C_VEL
LIN {X 0,Y 594.347,Z 321.451,A -85,B 0,C 180,E1 -1217.148,E2 -1217.148} C_VEL
LIN {X 0,Y 594.353,Z 321.453,A -85,B 0,C 180,E1 -1219.431,E2 -1219.431} C_VEL
LIN {X 0,Y 594.374,Z 321.441,A -85,B 0,C 180,E1 -1222.392,E2 -1222.392} C_VEL
LIN {X 0,Y 594.372,Z 321.45,A -85,B 0,C 180,E1 -1225.419,E2 -1225.419} C_VEL
LIN {X 0,Y 594.361,Z 321.443,A -85,B 0,C 180,E1 -1228.358,E2 -1228.358} C_VEL
LIN {X 0,Y 594.373,Z 321.449,A -85,B 0,C 180,E1 -1231.042,E2 -1231.042} C_VEL
LIN {X 0,Y 594.375,Z 321.449,A -85,B 0,C 180,E1 -1233.3,E2 -1233.3} C_VEL
LIN {X 0,Y 594.353,Z 321.444,A -85,B 0,C 180,E1 -1236.294,E2 -1236.294} C_VEL
LIN {X 0,Y 594.393,Z 321.447,A -85,B 0,C 180,E1 -1239.224,E2 -1239.224} C_VEL
LIN {X 0,Y 594.33,Z 321.447,A -85,B 0,C 180,E1 -1242.094,E2 -1242.094} C_VEL
LIN {X 0,Y 594.349,Z 321.445,A -85,B 0,C 180,E1 -1244.218,E2 -1244.218} C_VEL
LIN {X 0,Y 594.356,Z 321.454,A -85,B 0,C 180,E1 -1247.017,E2 -1247.017} C_VEL
LIN {X 0,Y 594.369,Z 321.442,A -85,B 0,C 180,E1 -1249.784,E2 -1249.784} C_VEL
LIN {X 0,Y 594.387,Z 321.444,A -85,B 0,C 180,E1 -1252.527,E2 -1252.527} C_VEL
LIN {X 0,Y 594.373,Z 321.445,A -85,B 0,C 180,E1 -1255.252,E2 -1255.252} C_VEL
LIN {X 0,Y 594.369,Z 321.442,A -85,B 0,C 180,E1 -1257.967,E2 -1257.967} C_VEL
LIN {X 0,Y 594.423,Z 321.444,A -85,B 0,C 180,E1 -1260.677,E2 -1260.677} C_VEL
LIN {X 0,Y 594.362,Z 321.444,A -85,B 0,C 180,E1 -1263.389,E2 -1263.389} C_VEL
LIN {X 0,Y 594.374,Z 321.442,A -85,B 0,C 180,E1 -1265.428,E2 -1265.428} C_VEL
LIN {X 0,Y 594.401,Z 321.44,A -85,B 0,C 180,E1 -1268.157,E2 -1268.157} C_VEL
LIN {X 0,Y 594.388,Z 321.443,A -85,B 0,C 180,E1 -1271.08,E2 -1271.08} C_VEL
LIN {X 0,Y 594.367,Z 321.442,A -85,B 0,C 180,E1 -1273.679,E2 -1273.679} C_VEL
LIN {X 0,Y 594.348,Z 321.445,A -85,B 0,C 180,E1 -1275.345,E2 -1275.345} C_VEL
LIN {X 0,Y 593.673,Z 321.53,A -85,B 0,C 180,E1 -1275.911,E2 -1275.911} C_VEL
LIN {X 0,Y 590.807,Z 321.891,A -85,B 0,C 180,E1 -1276.829,E2 -1276.829} C_VEL
LIN {X 0,Y 588.398,Z 322.191,A -85,B 0,C 180,E1 -1277.568,E2 -1277.568} C_VEL
LIN {X 0,Y 587.378,Z 322.316,A -85,B 0,C 180,E1 -1278.138,E2 -1278.138} C_VEL
LIN {X 0,Y 587.303,Z 322.325,A -85,B 0,C 180,E1 -1278.331,E2 -1278.331} C_VEL
LIN {X 0,Y 587.348,Z 322.319,A -85,B 0,C 180,E1 -1281.045,E2 -1281.045} C_VEL
LIN {X 0,Y 587.357,Z 322.316,A -85,B 0,C 180,E1 -1283.257,E2 -1283.257} C_VEL
LIN {X 0,Y 587.348,Z 322.322,A -85,B 0,C 180,E1 -1286.182,E2 -1286.182} C_VEL
LIN {X 0,Y 587.345,Z 322.318,A -85,B 0,C 180,E1 -1289.135,E2 -1289.135} C_VEL
LIN {X 0,Y 587.339,Z 322.32,A -85,B 0,C 180,E1 -1291.837,E2 -1291.837} C_VEL
LIN {X 0,Y 587.343,Z 322.327,A -85,B 0,C 180,E1 -1294.349,E2 -1294.349} C_VEL
LIN {X 0,Y 587.345,Z 322.32,A -85,B 0,C 180,E1 -1296.747,E2 -1296.747} C_VEL
LIN {X 0,Y 587.328,Z 322.319,A -85,B 0,C 180,E1 -1299.361,E2 -1299.361} C_VEL
LIN {X 0,Y 587.328,Z 322.327,A -85,B 0,C 180,E1 -1302.109,E2 -1302.109} C_VEL
LIN {X 0,Y 587.31,Z 322.321,A -85,B 0,C 180,E1 -1305.09,E2 -1305.09} C_VEL
LIN {X 0,Y 587.349,Z 322.323,A -85,B 0,C 180,E1 -1307.928,E2 -1307.928} C_VEL
LIN {X 0,Y 587.32,Z 322.32,A -85,B 0,C 180,E1 -1311.06,E2 -1311.06} C_VEL
LIN {X 0,Y 587.35,Z 322.317,A -85,B 0,C 180,E1 -1313.293,E2 -1313.293} C_VEL
LIN {X 0,Y 587.36,Z 322.321,A -85,B 0,C 180,E1 -1315.781,E2 -1315.781} C_VEL
LIN {X 0,Y 587.342,Z 322.323,A -85,B 0,C 180,E1 -1318.232,E2 -1318.232} C_VEL
LIN {X 0,Y 587.351,Z 322.316,A -85,B 0,C 180,E1 -1320.867,E2 -1320.867} C_VEL
LIN {X 0,Y 587.363,Z 322.323,A -85,B 0,C 180,E1 -1323.819,E2 -1323.819} C_VEL
LIN {X 0,Y 587.34,Z 322.326,A -85,B 0,C 180,E1 -1325.994,E2 -1325.994} C_VEL
LIN {X 0,Y 587.323,Z 322.324,A -85,B 0,C 180,E1 -1328.226,E2 -1328.226} C_VEL
LIN {X 0,Y 587.352,Z 322.317,A -85,B 0,C 180,E1 -1331.152,E2 -1331.152} C_VEL
LIN {X 0,Y 587.327,Z 322.325,A -85,B 0,C 180,E1 -1334.025,E2 -1334.025} C_VEL
LIN {X 0,Y 587.361,Z 322.318,A -85,B 0,C 180,E1 -1336.155,E2 -1336.155} C_VEL
LIN {X 0,Y 587.347,Z 322.317,A -85,B 0,C 180,E1 -1338.963,E2 -1338.963} C_VEL
LIN {X 0,Y 587.374,Z 322.322,A -85,B 0,C 180,E1 -1341.745,E2 -1341.745} C_VEL
LIN {X 0,Y 587.363,Z 322.315,A -85,B 0,C 180,E1 -1344.507,E2 -1344.507} C_VEL
LIN {X 0,Y 587.379,Z 322.317,A -85,B 0,C 180,E1 -1347.257,E2 -1347.257} C_VEL
LIN {X 0,Y 587.387,Z 322.315,A -85,B 0,C 180,E1 -1350,E2 -1350} C_VEL
LIN {X 0,Y 587.373,Z 322.314,A -85,B 0,C 180,E1 -1352.743,E2 -1352.743} C_VEL
LIN {X 0,Y 587.369,Z 322.324,A -85,B 0,C 180,E1 -1355.493,E2 -1355.493} C_VEL
LIN {X 0,Y 587.369,Z 322.314,A -85,B 0,C 180,E1 -1358.255,E2 -1358.255} C_VEL
LIN {X 0,Y 587.351,Z 322.322,A -85,B 0,C 180,E1 -1361.133,E2 -1361.133} C_VEL
LIN {X 0,Y 587.368,Z 322.314,A -85,B 0,C 180,E1 -1364.26,E2 -1364.26} C_VEL
LIN {X 0,Y 587.362,Z 322.323,A -85,B 0,C 180,E1 -1367.405,E2 -1367.405} C_VEL
LIN {X 0,Y 587.333,Z 322.318,A -85,B 0,C 180,E1 -1370.304,E2 -1370.304} C_VEL
LIN {X 0,Y 587.325,Z 322.329,A -85,B 0,C 180,E1 -1373.258,E2 -1373.258} C_VEL
LIN {X 0,Y 587.341,Z 322.322,A -85,B 0,C 180,E1 -1375.516,E2 -1375.516} C_VEL
LIN {X 0,Y 587.35,Z 322.317,A -85,B 0,C 180,E1 -1377.817,E2 -1377.817} C_VEL
LIN {X 0,Y 587.342,Z 322.319,A -85,B 0,C 180,E1 -1380.51,E2 -1380.51} C_VEL
LIN {X 0,Y 587.34,Z 322.328,A -85,B 0,C 180,E1 -1383.111,E2 -1383.111} C_VEL
LIN {X 0,Y 587.356,Z 322.316,A -85,B 0,C 180,E1 -1385.894,E2 -1385.894} C_VEL
LIN {X 0,Y 587.333,Z 322.321,A -85,B 0,C 180,E1 -1388.478,E2 -1388.478} C_VEL
LIN {X 0,Y 587.361,Z 322.322,A -85,B 0,C 180,E1 -1391.154,E2 -1391.154} C_VEL
LIN {X 0,Y 587.33,Z 322.32,A -85,B 0,C 180,E1 -1394.113,E2 -1394.113} C_VEL
LIN {X 0,Y 587.332,Z 322.328,A -85,B 0,C 180,E1 -1396.995,E2 -1396.995} C_VEL
LIN {X 0,Y 587.325,Z 322.316,A -85,B 0,C 180,E1 -1399.746,E2 -1399.746} C_VEL
LIN {X 0,Y 587.36,Z 322.339,A -85,B 0,C 180,E1 -1400.313,E2 -1400.313} C_VEL
LIN {X 0,Y 587.653,Z 328.712,A -85,B 0,C 180,E1 -1400.554,E2 -1400.554} C_VEL
LIN {X 0,Y 587.539,Z 340.78,A -85,B 0,C 180,E1 -1401.093,E2 -1401.093} C_VEL
LIN {X 0,Y 587.469,Z 351.678,A -85,B 0,C 180,E1 -1401.719,E2 -1401.719} C_VEL
LIN {X 0,Y 587.398,Z 361.247,A -85,B 0,C 180,E1 -1402.396,E2 -1402.396} C_VEL
LIN {X 0,Y 587.321,Z 371.137,A -85,B 0,C 180,E1 -1403.251,E2 -1403.251} C_VEL
LIN {X 0,Y 587.299,Z 379.198,A -85,B 0,C 180,E1 -1404.1,E2 -1404.1} C_VEL
LIN {X 0,Y 587.245,Z 387.158,A -85,B 0,C 180,E1 -1405.135,E2 -1405.135} C_VEL
LIN {X 0,Y 587.22,Z 392.509,A -85,B 0,C 180,E1 -1405.978,E2 -1405.978} C_VEL
LIN {X 0,Y 587.163,Z 397.4,A -85,B 0,C 180,E1 -1406.912,E2 -1406.912} C_VEL
LIN {X 0,Y 587.168,Z 401.236,A -85,B 0,C 180,E1 -1407.817,E2 -1407.817} C_VEL
LIN {X 0,Y 587.157,Z 405.053,A -85,B 0,C 180,E1 -1409.023,E2 -1409.023} C_VEL
LIN {X 0,Y 587.148,Z 406.862,A -85,B 0,C 180,E1 -1409.819,E2 -1409.819} C_VEL
LIN {X 0,Y 587.156,Z 408.393,A -85,B 0,C 180,E1 -1410.898,E2 -1410.898} C_VEL
LIN {X 0,Y 587.136,Z 408.81,A -85,B 0,C 180,E1 -1411.393,E2 -1411.393} C_VEL
LIN {X 0,Y 587.156,Z 408.95,A -85,B 0,C 180,E1 -1412.341,E2 -1412.341} C_VEL
LIN {X 0,Y 587.117,Z 407.799,A -85,B 0,C 180,E1 -1413.711,E2 -1413.711} C_VEL
LIN {X 0,Y 587.116,Z 406.492,A -85,B 0,C 180,E1 -1414.473,E2 -1414.473} C_VEL
LIN {X 0,Y 587.163,Z 404.022,A -85,B 0,C 180,E1 -1415.457,E2 -1415.457} C_VEL
LIN {X 0,Y 587.189,Z 399.383,A -85,B 0,C 180,E1 -1416.736,E2 -1416.736} C_VEL
LIN {X 0,Y 587.186,Z 393.963,A -85,B 0,C 180,E1 -1417.851,E2 -1417.851} C_VEL
LIN {X 0,Y 587.222,Z 388.371,A -85,B 0,C 180,E1 -1418.775,E2 -1418.775} C_VEL
LIN {X 0,Y 587.249,Z 381.64,A -85,B 0,C 180,E1 -1419.692,E2 -1419.692} C_VEL
LIN {X 0,Y 587.336,Z 372.195,A -85,B 0,C 180,E1 -1420.736,E2 -1420.736} C_VEL
LIN {X 0,Y 587.4,Z 363.516,A -85,B 0,C 180,E1 -1421.515,E2 -1421.515} C_VEL
LIN {X 0,Y 587.459,Z 353.713,A -85,B 0,C 180,E1 -1422.238,E2 -1422.238} C_VEL
LIN {X 0,Y 587.534,Z 343.835,A -85,B 0,C 180,E1 -1422.834,E2 -1422.834} C_VEL
LIN {X 0,Y 587.61,Z 332.894,A -85,B 0,C 180,E1 -1423.363,E2 -1423.363} C_VEL
LIN {X 0,Y 587.537,Z 323.258,A -85,B 0,C 180,E1 -1423.741,E2 -1423.741} C_VEL
LIN {X 0,Y 587.369,Z 322.362,A -85,B 0,C 180,E1 -1423.892,E2 -1423.892} C_VEL
LIN {X 0,Y 587.349,Z 322.319,A -85,B 0,C 180,E1 -1426.154,E2 -1426.154} C_VEL
LIN {X 0,Y 587.339,Z 322.322,A -85,B 0,C 180,E1 -1428.962,E2 -1428.962} C_VEL
LIN {X 0,Y 587.357,Z 322.32,A -85,B 0,C 180,E1 -1431.745,E2 -1431.745} C_VEL
LIN {X 0,Y 587.339,Z 322.318,A -85,B 0,C 180,E1 -1434.507,E2 -1434.507} C_VEL
LIN {X 0,Y 587.373,Z 322.323,A -85,B 0,C 180,E1 -1437.257,E2 -1437.257} C_VEL
LIN {X 0,Y 587.358,Z 322.316,A -85,B 0,C 180,E1 -1440,E2 -1440} C_VEL
LIN {X 0,Y 587.359,Z 322.318,A -85,B 0,C 180,E1 -1442.743,E2 -1442.743} C_VEL
LIN {X 0,Y 587.351,Z 322.322,A -85,B 0,C 180,E1 -1445.493,E2 -1445.493} C_VEL
LIN {X 0,Y 587.312,Z 322.321,A -85,B 0,C 180,E1 -1448.256,E2 -1448.256} C_VEL
LIN {X 0,Y 587.336,Z 322.329,A -85,B 0,C 180,E1 -1451.134,E2 -1451.134} C_VEL
LIN {X 0,Y 587.344,Z 322.317,A -85,B 0,C 180,E1 -1454.257,E2 -1454.257} C_VEL
LIN {X 0,Y 587.335,Z 322.322,A -85,B 0,C 180,E1 -1457.407,E2 -1457.407} C_VEL
LIN {X 0,Y 587.298,Z 322.325,A -85,B 0,C 180,E1 -1459.577,E2 -1459.577} C_VEL
LIN {X 0,Y 587.3,Z 322.323,A -85,B 0,C 180,E1 -1461.775,E2 -1461.775} C_VEL
LIN {X 0,Y 587.337,Z 322.324,A -85,B 0,C 180,E1 -1464.759,E2 -1464.759} C_VEL
LIN {X 0,Y 587.336,Z 322.318,A -85,B 0,C 180,E1 -1467.818,E2 -1467.818} C_VEL
LIN {X 0,Y 587.311,Z 322.325,A -85,B 0,C 180,E1 -1470.508,E2 -1470.508} C_VEL
LIN {X 0,Y 587.326,Z 322.326,A -85,B 0,C 180,E1 -1473.112,E2 -1473.112} C_VEL
LIN {X 0,Y 587.279,Z 322.325,A -85,B 0,C 180,E1 -1475.901,E2 -1475.901} C_VEL
LIN {X 0,Y 587.309,Z 322.327,A -85,B 0,C 180,E1 -1478.481,E2 -1478.481} C_VEL
LIN {X 0,Y 587.302,Z 322.326,A -85,B 0,C 180,E1 -1481.16,E2 -1481.16} C_VEL
LIN {X 0,Y 587.295,Z 322.325,A -85,B 0,C 180,E1 -1484.112,E2 -1484.112} C_VEL
LIN {X 0,Y 587.285,Z 322.33,A -85,B 0,C 180,E1 -1486.992,E2 -1486.992} C_VEL
LIN {X 0,Y 587.297,Z 322.324,A -85,B 0,C 180,E1 -1489.745,E2 -1489.745} C_VEL
LIN {X 0,Y 587.327,Z 322.328,A -85,B 0,C 180,E1 -1492.392,E2 -1492.392} C_VEL
LIN {X 0,Y 587.354,Z 322.511,A -85,B 0,C 180,E1 -1494.053,E2 -1494.053} C_VEL
LIN {X 0,Y 587.77,Z 325.599,A -85,B 0,C 180,E1 -1494.698,E2 -1494.698} C_VEL
LIN {X 0,Y 587.596,Z 339.88,A -85,B 0,C 180,E1 -1497.438,E2 -1497.438} C_VEL
LIN {X 0,Y 587.78,Z 355.023,A -85,B 0,C 180,E1 -1500.251,E2 -1500.251} C_VEL
LIN {X 0,Y 587.85,Z 365.908,A -85,B 0,C 180,E1 -1502.215,E2 -1502.215} C_VEL
LIN {X 0,Y 587.718,Z 379.585,A -85,B 0,C 180,E1 -1504.881,E2 -1504.881} C_VEL
LIN {X 0,Y 587.61,Z 393.279,A -85,B 0,C 180,E1 -1507.498,E2 -1507.498} C_VEL
LIN {X 0,Y 587.52,Z 406.974,A -85,B 0,C 180,E1 -1510.068,E2 -1510.068} C_VEL
LIN {X 0,Y 587.42,Z 420.669,A -85,B 0,C 180,E1 -1512.597,E2 -1512.597} C_VEL
LIN {X 0,Y 587.351,Z 436.32,A -85,B 0,C 180,E1 -1515.447,E2 -1515.447} C_VEL
LIN {X 0,Y 587.315,Z 449.055,A -85,B 0,C 180,E1 -1517.715,E2 -1517.715} C_VEL
LIN {X 0,Y 587.506,Z 450.748,A -85,B 0,C 180,E1 -1517.785,E2 -1517.785} C_VEL
LIN {X 0,Y 587.672,Z 463.29,A -85,B 0,C 180,E1 -1518.029,E2 -1518.029} C_VEL
LIN {X 0,Y 587.645,Z 475.954,A -85,B 0,C 180,E1 -1518.408,E2 -1518.408} C_VEL
LIN {X 0,Y 587.568,Z 487.915,A -85,B 0,C 180,E1 -1518.903,E2 -1518.903} C_VEL
LIN {X 0,Y 587.494,Z 500.176,A -85,B 0,C 180,E1 -1519.576,E2 -1519.576} C_VEL
LIN {X 0,Y 587.394,Z 511.393,A -85,B 0,C 180,E1 -1520.357,E2 -1520.357} C_VEL
LIN {X 0,Y 587.336,Z 521.346,A -85,B 0,C 180,E1 -1521.225,E2 -1521.225} C_VEL
LIN {X 0,Y 587.273,Z 530.951,A -85,B 0,C 180,E1 -1522.263,E2 -1522.263} C_VEL
LIN {X 0,Y 587.232,Z 537.461,A -85,B 0,C 180,E1 -1523.127,E2 -1523.127} C_VEL
LIN {X 0,Y 587.23,Z 543.869,A -85,B 0,C 180,E1 -1524.161,E2 -1524.161} C_VEL
LIN {X 0,Y 587.146,Z 548.956,A -85,B 0,C 180,E1 -1525.194,E2 -1525.194} C_VEL
LIN {X 0,Y 587.213,Z 552.898,A -85,B 0,C 180,E1 -1526.226,E2 -1526.226} C_VEL
LIN {X 0,Y 587.131,Z 555.807,A -85,B 0,C 180,E1 -1527.256,E2 -1527.256} C_VEL
LIN {X 0,Y 587.141,Z 557.203,A -85,B 0,C 180,E1 -1527.942,E2 -1527.942} C_VEL
LIN {X 0,Y 587.14,Z 558.784,A -85,B 0,C 180,E1 -1529.314,E2 -1529.314} C_VEL
LIN {X 0,Y 587.137,Z 559,A -85,B 0,C 180,E1 -1530,E2 -1530} C_VEL
LIN {X 0,Y 587.147,Z 558.186,A -85,B 0,C 180,E1 -1531.372,E2 -1531.372} C_VEL
LIN {X 0,Y 587.141,Z 557.203,A -85,B 0,C 180,E1 -1532.058,E2 -1532.058} C_VEL
LIN {X 0,Y 587.131,Z 555.807,A -85,B 0,C 180,E1 -1532.744,E2 -1532.744} C_VEL
LIN {X 0,Y 587.213,Z 552.898,A -85,B 0,C 180,E1 -1533.774,E2 -1533.774} C_VEL
LIN {X 0,Y 587.146,Z 548.955,A -85,B 0,C 180,E1 -1534.806,E2 -1534.806} C_VEL
LIN {X 0,Y 587.23,Z 543.869,A -85,B 0,C 180,E1 -1535.839,E2 -1535.839} C_VEL
LIN {X 0,Y 587.232,Z 537.461,A -85,B 0,C 180,E1 -1536.873,E2 -1536.873} C_VEL
LIN {X 0,Y 587.287,Z 529.48,A -85,B 0,C 180,E1 -1537.91,E2 -1537.91} C_VEL
LIN {X 0,Y 587.336,Z 521.346,A -85,B 0,C 180,E1 -1538.775,E2 -1538.775} C_VEL
LIN {X 0,Y 587.393,Z 511.393,A -85,B 0,C 180,E1 -1539.643,E2 -1539.643} C_VEL
LIN {X 0,Y 587.494,Z 500.177,A -85,B 0,C 180,E1 -1540.424,E2 -1540.424} C_VEL
LIN {X 0,Y 587.571,Z 489.201,A -85,B 0,C 180,E1 -1541.033,E2 -1541.033} C_VEL
LIN {X 0,Y 587.602,Z 477.209,A -85,B 0,C 180,E1 -1541.549,E2 -1541.549} C_VEL
LIN {X 0,Y 587.691,Z 464.161,A -85,B 0,C 180,E1 -1541.948,E2 -1541.948} C_VEL
LIN {X 0,Y 587.637,Z 451.533,A -85,B 0,C 180,E1 -1542.2,E2 -1542.2} C_VEL
LIN {X 0,Y 587.349,Z 449.31,A -85,B 0,C 180,E1 -1542.262,E2 -1542.262} C_VEL
LIN {X 0,Y 587.281,Z 444.145,A -85,B 0,C 180,E1 -1543.142,E2 -1543.142} C_VEL
LIN {X 0,Y 587.361,Z 430.45,A -85,B 0,C 180,E1 -1545.618,E2 -1545.618} C_VEL
LIN {X 0,Y 587.476,Z 414.799,A -85,B 0,C 180,E1 -1548.482,E2 -1548.482} C_VEL
LIN {X 0,Y 587.569,Z 399.15,A -85,B 0,C 180,E1 -1551.395,E2 -1551.395} C_VEL
LIN {X 0,Y 587.695,Z 385.454,A -85,B 0,C 180,E1 -1553.99,E2 -1553.99} C_VEL
LIN {X 0,Y 587.798,Z 371.761,A -85,B 0,C 180,E1 -1556.638,E2 -1556.638} C_VEL
LIN {X 0,Y 587.827,Z 359.984,A -85,B 0,C 180,E1 -1558.892,E2 -1558.892} C_VEL
LIN {X 0,Y 587.785,Z 346.092,A -85,B 0,C 180,E1 -1561.54,E2 -1561.54} C_VEL
LIN {X 0,Y 587.908,Z 331.449,A -85,B 0,C 180,E1 -1564.427,E2 -1564.427} C_VEL
LIN {X 0,Y 587.776,Z 324.489,A -85,B 0,C 180,E1 -1565.865,E2 -1565.865} C_VEL
LIN {X 0,Y 587.327,Z 322.46,A -85,B 0,C 180,E1 -1566.321,E2 -1566.321} C_VEL
LIN {X 0,Y 587.298,Z 322.327,A -85,B 0,C 180,E1 -1568.937,E2 -1568.937} C_VEL
LIN {X 0,Y 587.328,Z 322.325,A -85,B 0,C 180,E1 -1571.156,E2 -1571.156} C_VEL
LIN {X 0,Y 587.306,Z 322.324,A -85,B 0,C 180,E1 -1574.111,E2 -1574.111} C_VEL
LIN {X 0,Y 587.296,Z 322.327,A -85,B 0,C 180,E1 -1576.992,E2 -1576.992} C_VEL
LIN {X 0,Y 587.297,Z 322.327,A -85,B 0,C 180,E1 -1579.744,E2 -1579.744} C_VEL
LIN {X 0,Y 587.329,Z 322.319,A -85,B 0,C 180,E1 -1582.391,E2 -1582.391} C_VEL
LIN {X 0,Y 587.331,Z 322.323,A -85,B 0,C 180,E1 -1585.653,E2 -1585.653} C_VEL
LIN {X 0,Y 587.326,Z 322.319,A -85,B 0,C 180,E1 -1588.23,E2 -1588.23} C_VEL
LIN {X 0,Y 587.337,Z 322.322,A -85,B 0,C 180,E1 -1590.866,E2 -1590.866} C_VEL
LIN {X 0,Y 587.322,Z 322.322,A -85,B 0,C 180,E1 -1593.72,E2 -1593.72} C_VEL
LIN {X 0,Y 587.302,Z 322.322,A -85,B 0,C 180,E1 -1595.992,E2 -1595.992} C_VEL
LIN {X 0,Y 587.319,Z 322.328,A -85,B 0,C 180,E1 -1598.962,E2 -1598.962} C_VEL
LIN {X 0,Y 587.337,Z 322.327,A -85,B 0,C 180,E1 -1601.151,E2 -1601.151} C_VEL
LIN {X 0,Y 587.305,Z 322.322,A -85,B 0,C 180,E1 -1604.024,E2 -1604.024} C_VEL
LIN {X 0,Y 587.338,Z 322.318,A -85,B 0,C 180,E1 -1606.154,E2 -1606.154} C_VEL
LIN {X 0,Y 587.332,Z 322.329,A -85,B 0,C 180,E1 -1608.962,E2 -1608.962} C_VEL
LIN {X 0,Y 587.312,Z 322.321,A -85,B 0,C 180,E1 -1611.744,E2 -1611.744} C_VEL
LIN {X 0,Y 587.351,Z 322.32,A -85,B 0,C 180,E1 -1614.507,E2 -1614.507} C_VEL
LIN {X 0,Y 587.359,Z 322.319,A -85,B 0,C 180,E1 -1617.257,E2 -1617.257} C_VEL
LIN {X 0,Y 587.358,Z 322.316,A -85,B 0,C 180,E1 -1620,E2 -1620} C_VEL
LIN {X 0,Y 587.373,Z 322.324,A -85,B 0,C 180,E1 -1622.743,E2 -1622.743} C_VEL
LIN {X 0,Y 587.339,Z 322.318,A -85,B 0,C 180,E1 -1625.493,E2 -1625.493} C_VEL
LIN {X 0,Y 587.357,Z 322.319,A -85,B 0,C 180,E1 -1628.255,E2 -1628.255} C_VEL
LIN {X 0,Y 587.351,Z 322.319,A -85,B 0,C 180,E1 -1631.142,E2 -1631.142} C_VEL
LIN {X 0,Y 587.353,Z 322.32,A -85,B 0,C 180,E1 -1634.261,E2 -1634.261} C_VEL
LIN {X 0,Y 587.338,Z 322.318,A -85,B 0,C 180,E1 -1637.406,E2 -1637.406} C_VEL
LIN {X 0,Y 587.303,Z 322.325,A -85,B 0,C 180,E1 -1638.331,E2 -1638.331} C_VEL
LIN {X 0,Y 586.662,Z 322.407,A -85,B 0,C 180,E1 -1638.903,E2 -1638.903} C_VEL
LIN {X 0,Y 583.834,Z 322.757,A -85,B 0,C 180,E1 -1639.832,E2 -1639.832} C_VEL
LIN {X 0,Y 581.421,Z 323.064,A -85,B 0,C 180,E1 -1640.579,E2 -1640.579} C_VEL
LIN {X 0,Y 580.371,Z 323.188,A -85,B 0,C 180,E1 -1641.155,E2 -1641.155} C_VEL
LIN {X 0,Y 580.278,Z 323.197,A -85,B 0,C 180,E1 -1641.35,E2 -1641.35} C_VEL
LIN {X 0,Y 580.293,Z 323.195,A -85,B 0,C 180,E1 -1643.557,E2 -1643.557} C_VEL
LIN {X 0,Y 580.281,Z 323.205,A -85,B 0,C 180,E1 -1646.335,E2 -1646.335} C_VEL
LIN {X 0,Y 580.289,Z 323.198,A -85,B 0,C 180,E1 -1648.976,E2 -1648.976} C_VEL
LIN {X 0,Y 580.271,Z 323.198,A -85,B 0,C 180,E1 -1651.386,E2 -1651.386} C_VEL
LIN {X 0,Y 580.309,Z 323.196,A -85,B 0,C 180,E1 -1653.855,E2 -1653.855} C_VEL
LIN {X 0,Y 580.294,Z 323.196,A -85,B 0,C 180,E1 -1656.936,E2 -1656.936} C_VEL
LIN {X 0,Y 580.284,Z 323.201,A -85,B 0,C 180,E1 -1659.934,E2 -1659.934} C_VEL
LIN {X 0,Y 580.272,Z 323.201,A -85,B 0,C 180,E1 -1662.707,E2 -1662.707} C_VEL
LIN {X 0,Y 580.269,Z 323.2,A -85,B 0,C 180,E1 -1665.609,E2 -1665.609} C_VEL
LIN {X 0,Y 580.31,Z 323.202,A -85,B 0,C 180,E1 -1668.235,E2 -1668.235} C_VEL
LIN {X 0,Y 580.275,Z 323.198,A -85,B 0,C 180,E1 -1670.966,E2 -1670.966} C_VEL
LIN {X 0,Y 580.29,Z 323.199,A -85,B 0,C 180,E1 -1673.599,E2 -1673.599} C_VEL
LIN {X 0,Y 580.304,Z 323.195,A -85,B 0,C 180,E1 -1676.684,E2 -1676.684} C_VEL
LIN {X 0,Y 580.301,Z 323.196,A -85,B 0,C 180,E1 -1679.426,E2 -1679.426} C_VEL
LIN {X 0,Y 580.32,Z 323.199,A -85,B 0,C 180,E1 -1682.138,E2 -1682.138} C_VEL
LIN {X 0,Y 580.309,Z 323.193,A -85,B 0,C 180,E1 -1684.921,E2 -1684.921} C_VEL
LIN {X 0,Y 580.274,Z 323.206,A -85,B 0,C 180,E1 -1687.948,E2 -1687.948} C_VEL
LIN {X 0,Y 580.321,Z 323.192,A -85,B 0,C 180,E1 -1690.915,E2 -1690.915} C_VEL
LIN {X 0,Y 580.282,Z 323.206,A -85,B 0,C 180,E1 -1693.826,E2 -1693.826} C_VEL
LIN {X 0,Y 580.328,Z 323.197,A -85,B 0,C 180,E1 -1695.983,E2 -1695.983} C_VEL
LIN {X 0,Y 580.308,Z 323.194,A -85,B 0,C 180,E1 -1698.827,E2 -1698.827} C_VEL
LIN {X 0,Y 580.337,Z 323.2,A -85,B 0,C 180,E1 -1701.644,E2 -1701.644} C_VEL
LIN {X 0,Y 580.33,Z 323.191,A -85,B 0,C 180,E1 -1704.44,E2 -1704.44} C_VEL
LIN {X 0,Y 580.347,Z 323.193,A -85,B 0,C 180,E1 -1707.918,E2 -1707.918} C_VEL
LIN {X 0,Y 580.362,Z 323.187,A -85,B 0,C 180,E1 -1710.694,E2 -1710.694} C_VEL
LIN {X 0,Y 580.292,Z 323.206,A -85,B 0,C 180,E1 -1713.472,E2 -1713.472} C_VEL
LIN {X 0,Y 580.336,Z 323.199,A -85,B 0,C 180,E1 -1715.56,E2 -1715.56} C_VEL
LIN {X 0,Y 580.331,Z 323.19,A -85,B 0,C 180,E1 -1718.356,E2 -1718.356} C_VEL
LIN {X 0,Y 580.303,Z 323.201,A -85,B 0,C 180,E1 -1721.191,E2 -1721.191} C_VEL
LIN {X 0,Y 580.33,Z 323.192,A -85,B 0,C 180,E1 -1724.016,E2 -1724.016} C_VEL
LIN {X 0,Y 580.314,Z 323.197,A -85,B 0,C 180,E1 -1726.913,E2 -1726.913} C_VEL
LIN {X 0,Y 580.308,Z 323.195,A -85,B 0,C 180,E1 -1729.822,E2 -1729.822} C_VEL
LIN {X 0,Y 580.297,Z 323.198,A -85,B 0,C 180,E1 -1732.802,E2 -1732.802} C_VEL
LIN {X 0,Y 580.31,Z 323.202,A -85,B 0,C 180,E1 -1735.079,E2 -1735.079} C_VEL
LIN {X 0,Y 580.321,Z 323.193,A -85,B 0,C 180,E1 -1737.862,E2 -1737.862} C_VEL
LIN {X 0,Y 580.292,Z 323.199,A -85,B 0,C 180,E1 -1740.695,E2 -1740.695} C_VEL
LIN {X 0,Y 580.304,Z 323.2,A -85,B 0,C 180,E1 -1743.316,E2 -1743.316} C_VEL
LIN {X 0,Y 580.325,Z 323.192,A -85,B 0,C 180,E1 -1745.767,E2 -1745.767} C_VEL
LIN {X 0,Y 580.288,Z 323.196,A -85,B 0,C 180,E1 -1748.145,E2 -1748.145} C_VEL
LIN {X 0,Y 580.318,Z 323.201,A -85,B 0,C 180,E1 -1750.841,E2 -1750.841} C_VEL
LIN {X 0,Y 580.287,Z 323.198,A -85,B 0,C 180,E1 -1753.656,E2 -1753.656} C_VEL
LIN {X 0,Y 580.287,Z 323.203,A -85,B 0,C 180,E1 -1756.607,E2 -1756.607} C_VEL
LIN {X 0,Y 580.316,Z 323.193,A -85,B 0,C 180,E1 -1759.158,E2 -1759.158} C_VEL
LIN {X 0,Y 580.32,Z 323.35,A -85,B 0,C 180,E1 -1760.216,E2 -1760.216} C_VEL
LIN {X 0,Y 580.695,Z 327.265,A -85,B 0,C 180,E1 -1760.36,E2 -1760.36} C_VEL
LIN {X 0,Y 580.571,Z 339.897,A -85,B 0,C 180,E1 -1760.915,E2 -1760.915} C_VEL
LIN {X 0,Y 580.505,Z 350.86,A -85,B 0,C 180,E1 -1761.539,E2 -1761.539} C_VEL
LIN {X 0,Y 580.368,Z 361.534,A -85,B 0,C 180,E1 -1762.3,E2 -1762.3} C_VEL
LIN {X 0,Y 580.305,Z 370.298,A -85,B 0,C 180,E1 -1763.063,E2 -1763.063} C_VEL
LIN {X 0,Y 580.23,Z 378.721,A -85,B 0,C 180,E1 -1763.95,E2 -1763.95} C_VEL
LIN {X 0,Y 580.169,Z 387.388,A -85,B 0,C 180,E1 -1765.084,E2 -1765.084} C_VEL
LIN {X 0,Y 580.129,Z 391.912,A -85,B 0,C 180,E1 -1765.794,E2 -1765.794} C_VEL
LIN {X 0,Y 580.089,Z 396.793,A -85,B 0,C 180,E1 -1766.714,E2 -1766.714} C_VEL
LIN {X 0,Y 580.077,Z 401.309,A -85,B 0,C 180,E1 -1767.786,E2 -1767.786} C_VEL
LIN {X 0,Y 580.064,Z 404.029,A -85,B 0,C 180,E1 -1768.602,E2 -1768.602} C_VEL
LIN {X 0,Y 580.064,Z 406.13,A -85,B 0,C 180,E1 -1769.411,E2 -1769.411} C_VEL
LIN {X 0,Y 580.061,Z 408.26,A -85,B 0,C 180,E1 -1770.73,E2 -1770.73} C_VEL
LIN {X 0,Y 580.044,Z 408.962,A -85,B 0,C 180,E1 -1772.186,E2 -1772.186} C_VEL
LIN {X 0,Y 580.036,Z 407.834,A -85,B 0,C 180,E1 -1773.714,E2 -1773.714} C_VEL
LIN {X 0,Y 580.066,Z 404.501,A -85,B 0,C 180,E1 -1775.322,E2 -1775.322} C_VEL
LIN {X 0,Y 580.088,Z 400.868,A -85,B 0,C 180,E1 -1776.434,E2 -1776.434} C_VEL
LIN {X 0,Y 580.106,Z 395.878,A -85,B 0,C 180,E1 -1777.566,E2 -1777.566} C_VEL
LIN {X 0,Y 580.167,Z 390.648,A -85,B 0,C 180,E1 -1778.504,E2 -1778.504} C_VEL
LIN {X 0,Y 580.23,Z 384.334,A -85,B 0,C 180,E1 -1779.436,E2 -1779.436} C_VEL
LIN {X 0,Y 580.273,Z 376.743,A -85,B 0,C 180,E1 -1780.361,E2 -1780.361} C_VEL
LIN {X 0,Y 580.316,Z 367.582,A -85,B 0,C 180,E1 -1781.281,E2 -1781.281} C_VEL
LIN {X 0,Y 580.427,Z 356.137,A -85,B 0,C 180,E1 -1782.198,E2 -1782.198} C_VEL
LIN {X 0,Y 580.541,Z 345.183,A -85,B 0,C 180,E1 -1782.891,E2 -1782.891} C_VEL
LIN {X 0,Y 580.639,Z 333.5,A -85,B 0,C 180,E1 -1783.474,E2 -1783.474} C_VEL
LIN {X 0,Y 580.587,Z 324.498,A -85,B 0,C 180,E1 -1783.834,E2 -1783.834} C_VEL
LIN {X 0,Y 580.332,Z 323.373,A -85,B 0,C 180,E1 -1783.962,E2 -1783.962} C_VEL
LIN {X 0,Y 580.267,Z 323.201,A -85,B 0,C 180,E1 -1786.696,E2 -1786.696} C_VEL
LIN {X 0,Y 580.293,Z 323.205,A -85,B 0,C 180,E1 -1789.533,E2 -1789.533} C_VEL
LIN {X 0,Y 580.316,Z 323.193,A -85,B 0,C 180,E1 -1792.344,E2 -1792.344} C_VEL
LIN {X 0,Y 580.331,Z 323.198,A -85,B 0,C 180,E1 -1795.137,E2 -1795.137} C_VEL
LIN {X 0,Y 580.316,Z 323.195,A -85,B 0,C 180,E1 -1797.918,E2 -1797.918} C_VEL
LIN {X 0,Y 580.328,Z 323.192,A -85,B 0,C 180,E1 -1800,E2 -1800} C_VEL
LIN {X 0,Y 580.326,Z 323.194,A -85,B 0,C 180,E1 -1802.777,E2 -1802.777} C_VEL
LIN {X 0,Y 580.314,Z 323.198,A -85,B 0,C 180,E1 -1805.56,E2 -1805.56} C_VEL
LIN {X 0,Y 580.31,Z 323.196,A -85,B 0,C 180,E1 -1807.656,E2 -1807.656} C_VEL
LIN {X 0,Y 580.283,Z 323.198,A -85,B 0,C 180,E1 -1810.467,E2 -1810.467} C_VEL
LIN {X 0,Y 580.26,Z 323.207,A -85,B 0,C 180,E1 -1813.304,E2 -1813.304} C_VEL
LIN {X 0,Y 580.28,Z 323.202,A -85,B 0,C 180,E1 -1815.453,E2 -1815.453} C_VEL
LIN {X 0,Y 580.277,Z 323.199,A -85,B 0,C 180,E1 -1817.625,E2 -1817.625} C_VEL
LIN {X 0,Y 580.273,Z 323.198,A -85,B 0,C 180,E1 -1819.824,E2 -1819.824} C_VEL
LIN {X 0,Y 580.245,Z 323.202,A -85,B 0,C 180,E1 -1822.054,E2 -1822.054} C_VEL
LIN {X 0,Y 580.29,Z 323.204,A -85,B 0,C 180,E1 -1825.081,E2 -1825.081} C_VEL
LIN {X 0,Y 580.288,Z 323.197,A -85,B 0,C 180,E1 -1828.186,E2 -1828.186} C_VEL
LIN {X 0,Y 580.262,Z 323.207,A -85,B 0,C 180,E1 -1830.693,E2 -1830.693} C_VEL
LIN {X 0,Y 580.271,Z 323.202,A -85,B 0,C 180,E1 -1833.314,E2 -1833.314} C_VEL
LIN {X 0,Y 580.234,Z 323.203,A -85,B 0,C 180,E1 -1835.757,E2 -1835.757} C_VEL
LIN {X 0,Y 580.274,Z 323.2,A -85,B 0,C 180,E1 -1838.148,E2 -1838.148} C_VEL
LIN {X 0,Y 580.272,Z 323.207,A -85,B 0,C 180,E1 -1840.846,E2 -1840.846} C_VEL
LIN {X 0,Y 580.235,Z 323.205,A -85,B 0,C 180,E1 -1843.388,E2 -1843.388} C_VEL
LIN {X 0,Y 580.262,Z 323.205,A -85,B 0,C 180,E1 -1846.342,E2 -1846.342} C_VEL
LIN {X 0,Y 580.289,Z 323.2,A -85,B 0,C 180,E1 -1849.157,E2 -1849.157} C_VEL
LIN {X 0,Y 580.272,Z 323.202,A -85,B 0,C 180,E1 -1851.93,E2 -1851.93} C_VEL
LIN {X 0,Y 580.287,Z 323.435,A -85,B 0,C 180,E1 -1853.889,E2 -1853.889} C_VEL
LIN {X 0,Y 580.822,Z 327.301,A -85,B 0,C 180,E1 -1854.707,E2 -1854.707} C_VEL
LIN {X 0,Y 580.644,Z 341.199,A -85,B 0,C 180,E1 -1857.411,E2 -1857.411} C_VEL
LIN {X 0,Y 580.786,Z 356.328,A -85,B 0,C 180,E1 -1860.256,E2 -1860.256} C_VEL
LIN {X 0,Y 580.842,Z 371.529,A -85,B 0,C 180,E1 -1863.017,E2 -1863.017} C_VEL
LIN {X 0,Y 580.762,Z 384.084,A -85,B 0,C 180,E1 -1865.438,E2 -1865.438} C_VEL
LIN {X 0,Y 580.609,Z 399.149,A -85,B 0,C 180,E1 -1868.335,E2 -1868.335} C_VEL
LIN {X 0,Y 580.48,Z 414.799,A -85,B 0,C 180,E1 -1871.287,E2 -1871.287} C_VEL
LIN {X 0,Y 580.344,Z 430.45,A -85,B 0,C 180,E1 -1874.189,E2 -1874.189} C_VEL
LIN {X 0,Y 580.247,Z 444.145,A -85,B 0,C 180,E1 -1876.696,E2 -1876.696} C_VEL
LIN {X 0,Y 580.26,Z 449.317,A -85,B 0,C 180,E1 -1877.586,E2 -1877.586} C_VEL
LIN {X 0,Y 580.783,Z 453.549,A -85,B 0,C 180,E1 -1877.686,E2 -1877.686} C_VEL
LIN {X 0,Y 580.763,Z 466.762,A -85,B 0,C 180,E1 -1877.973,E2 -1877.973} C_VEL
LIN {X 0,Y 580.66,Z 479.268,A -85,B 0,C 180,E1 -1878.392,E2 -1878.392} C_VEL
LIN {X 0,Y 580.57,Z 490.919,A -85,B 0,C 180,E1 -1878.921,E2 -1878.921} C_VEL
LIN {X 0,Y 580.461,Z 502.938,A -85,B 0,C 180,E1 -1879.625,E2 -1879.625} C_VEL
LIN {X 0,Y 580.364,Z 513.545,A -85,B 0,C 180,E1 -1880.415,E2 -1880.415} C_VEL
LIN {X 0,Y 580.262,Z 523.101,A -85,B 0,C 180,E1 -1881.292,E2 -1881.292} C_VEL
LIN {X 0,Y 580.221,Z 530.95,A -85,B 0,C 180,E1 -1882.168,E2 -1882.168} C_VEL
LIN {X 0,Y 580.157,Z 538.659,A -85,B 0,C 180,E1 -1883.222,E2 -1883.222} C_VEL
LIN {X 0,Y 580.138,Z 545.677,A -85,B 0,C 180,E1 -1884.439,E2 -1884.439} C_VEL
LIN {X 0,Y 580.108,Z 550.368,A -85,B 0,C 180,E1 -1885.484,E2 -1885.484} C_VEL
LIN {X 0,Y 580.123,Z 553.955,A -85,B 0,C 180,E1 -1886.527,E2 -1886.527} C_VEL
LIN {X 0,Y 580.043,Z 555.807,A -85,B 0,C 180,E1 -1887.222,E2 -1887.222} C_VEL
LIN {X 0,Y 580.04,Z 557.202,A -85,B 0,C 180,E1 -1887.917,E2 -1887.917} C_VEL
LIN {X 0,Y 580.04,Z 558.784,A -85,B 0,C 180,E1 -1889.306,E2 -1889.306} C_VEL
LIN {X 0,Y 580.037,Z 559,A -85,B 0,C 180,E1 -1890,E2 -1890} C_VEL
LIN {X 0,Y 580.046,Z 558.186,A -85,B 0,C 180,E1 -1891.389,E2 -1891.389} C_VEL
LIN {X 0,Y 580.04,Z 557.203,A -85,B 0,C 180,E1 -1892.083,E2 -1892.083} C_VEL
LIN {X 0,Y 580.043,Z 555.808,A -85,B 0,C 180,E1 -1892.778,E2 -1892.778} C_VEL
LIN {X 0,Y 580.109,Z 552.898,A -85,B 0,C 180,E1 -1893.82,E2 -1893.82} C_VEL
LIN {X 0,Y 580.053,Z 548.955,A -85,B 0,C 180,E1 -1894.865,E2 -1894.865} C_VEL
LIN {X 0,Y 580.162,Z 543.869,A -85,B 0,C 180,E1 -1895.91,E2 -1895.91} C_VEL
LIN {X 0,Y 580.159,Z 537.461,A -85,B 0,C 180,E1 -1896.958,E2 -1896.958} C_VEL
LIN {X 0,Y 580.241,Z 529.481,A -85,B 0,C 180,E1 -1898.007,E2 -1898.007} C_VEL
LIN {X 0,Y 580.305,Z 521.346,A -85,B 0,C 180,E1 -1898.883,E2 -1898.883} C_VEL
LIN {X 0,Y 580.375,Z 511.394,A -85,B 0,C 180,E1 -1899.76,E2 -1899.76} C_VEL
LIN {X 0,Y 580.499,Z 500.178,A -85,B 0,C 180,E1 -1900.551,E2 -1900.551} C_VEL
LIN {X 0,Y 580.588,Z 489.2,A -85,B 0,C 180,E1 -1901.167,E2 -1901.167} C_VEL
LIN {X 0,Y 580.654,Z 476.99,A -85,B 0,C 180,E1 -1901.696,E2 -1901.696} C_VEL
LIN {X 0,Y 580.729,Z 464.161,A -85,B 0,C 180,E1 -1902.094,E2 -1902.094} C_VEL
LIN {X 0,Y 580.612,Z 451.622,A -85,B 0,C 180,E1 -1902.348,E2 -1902.348} C_VEL
LIN {X 0,Y 580.26,Z 449.305,A -85,B 0,C 180,E1 -1902.414,E2 -1902.414} C_VEL
LIN {X 0,Y 580.303,Z 442.189,A -85,B 0,C 180,E1 -1903.66,E2 -1903.66} C_VEL
LIN {X 0,Y 580.384,Z 426.538,A -85,B 0,C 180,E1 -1906.533,E2 -1906.533} C_VEL
LIN {X 0,Y 580.487,Z 412.182,A -85,B 0,C 180,E1 -1909.204,E2 -1909.204} C_VEL
LIN {X 0,Y 580.626,Z 397.192,A -85,B 0,C 180,E1 -1912.038,E2 -1912.038} C_VEL
LIN {X 0,Y 580.781,Z 382.715,A -85,B 0,C 180,E1 -1914.828,E2 -1914.828} C_VEL
LIN {X 0,Y 580.852,Z 370.547,A -85,B 0,C 180,E1 -1917.177,E2 -1917.177} C_VEL
LIN {X 0,Y 580.868,Z 355.927,A -85,B 0,C 180,E1 -1919.939,E2 -1919.939} C_VEL
LIN {X 0,Y 580.886,Z 340.427,A -85,B 0,C 180,E1 -1922.986,E2 -1922.986} C_VEL
LIN {X 0,Y 581.066,Z 328.153,A -85,B 0,C 180,E1 -1925.489,E2 -1925.489} C_VEL
LIN {X 0,Y 580.281,Z 323.29,A -85,B 0,C 180,E1 -1926.591,E2 -1926.591} C_VEL
LIN {X 0,Y 580.276,Z 323.205,A -85,B 0,C 180,E1 -1929.182,E2 -1929.182} C_VEL
LIN {X 0,Y 580.245,Z 323.208,A -85,B 0,C 180,E1 -1931.771,E2 -1931.771} C_VEL
LIN {X 0,Y 580.242,Z 323.203,A -85,B 0,C 180,E1 -1934.627,E2 -1934.627} C_VEL
LIN {X 0,Y 580.277,Z 323.204,A -85,B 0,C 180,E1 -1937.628,E2 -1937.628} C_VEL
LIN {X 0,Y 580.268,Z 323.199,A -85,B 0,C 180,E1 -1940.065,E2 -1940.065} C_VEL
LIN {X 0,Y 580.289,Z 323.202,A -85,B 0,C 180,E1 -1943.065,E2 -1943.065} C_VEL
LIN {X 0,Y 580.27,Z 323.198,A -85,B 0,C 180,E1 -1946.142,E2 -1946.142} C_VEL
LIN {X 0,Y 580.259,Z 323.201,A -85,B 0,C 180,E1 -1948.613,E2 -1948.613} C_VEL
LIN {X 0,Y 580.28,Z 323.204,A -85,B 0,C 180,E1 -1951.023,E2 -1951.023} C_VEL
LIN {X 0,Y 580.276,Z 323.2,A -85,B 0,C 180,E1 -1953.666,E2 -1953.666} C_VEL
LIN {X 0,Y 580.279,Z 323.199,A -85,B 0,C 180,E1 -1955.683,E2 -1955.683} C_VEL
LIN {X 0,Y 580.245,Z 323.201,A -85,B 0,C 180,E1 -1957.946,E2 -1957.946} C_VEL
LIN {X 0,Y 580.288,Z 323.203,A -85,B 0,C 180,E1 -1960.913,E2 -1960.913} C_VEL
LIN {X 0,Y 580.26,Z 323.2,A -85,B 0,C 180,E1 -1963.825,E2 -1963.825} C_VEL
LIN {X 0,Y 580.305,Z 323.194,A -85,B 0,C 180,E1 -1965.982,E2 -1965.982} C_VEL
LIN {X 0,Y 580.293,Z 323.203,A -85,B 0,C 180,E1 -1968.827,E2 -1968.827} C_VEL
LIN {X 0,Y 580.286,Z 323.197,A -85,B 0,C 180,E1 -1971.643,E2 -1971.643} C_VEL
LIN {X 0,Y 580.256,Z 323.2,A -85,B 0,C 180,E1 -1973.742,E2 -1973.742} C_VEL
LIN {X 0,Y 580.242,Z 323.202,A -85,B 0,C 180,E1 -1975.832,E2 -1975.832} C_VEL
LIN {X 0,Y 580.313,Z 323.193,A -85,B 0,C 180,E1 -1977.918,E2 -1977.918} C_VEL
LIN {X 0,Y 580.361,Z 323.195,A -85,B 0,C 180,E1 -1980.694,E2 -1980.694} C_VEL
LIN {X 0,Y 580.265,Z 323.2,A -85,B 0,C 180,E1 -1983.472,E2 -1983.472} C_VEL
LIN {X 0,Y 580.305,Z 323.194,A -85,B 0,C 180,E1 -1985.56,E2 -1985.56} C_VEL
LIN {X 0,Y 580.321,Z 323.197,A -85,B 0,C 180,E1 -1988.356,E2 -1988.356} C_VEL
LIN {X 0,Y 580.322,Z 323.194,A -85,B 0,C 180,E1 -1991.209,E2 -1991.209} C_VEL
LIN {X 0,Y 580.303,Z 323.2,A -85,B 0,C 180,E1 -1994.339,E2 -1994.339} C_VEL
LIN {X 0,Y 580.304,Z 323.198,A -85,B 0,C 180,E1 -1996.915,E2 -1996.915} C_VEL
LIN {X 0,Y 580.297,Z 323.196,A -85,B 0,C 180,E1 -1999.823,E2 -1999.823} C_VEL
LIN {X 0,Y 580.278,Z 323.197,A -85,B 0,C 180,E1 -2001.35,E2 -2001.35} C_VEL
LIN {X 0,Y 579.588,Z 323.286,A -85,B 0,C 180,E1 -2001.93,E2 -2001.93} C_VEL
LIN {X 0,Y 576.716,Z 323.645,A -85,B 0,C 180,E1 -2002.87,E2 -2002.87} C_VEL
LIN {X 0,Y 574.319,Z 323.941,A -85,B 0,C 180,E1 -2003.627,E2 -2003.627} C_VEL
LIN {X 0,Y 573.315,Z 324.07,A -85,B 0,C 180,E1 -2004.211,E2 -2004.211} C_VEL
LIN {X 0,Y 573.245,Z 324.077,A -85,B 0,C 180,E1 -2004.408,E2 -2004.408} C_VEL
LIN {X 0,Y 573.241,Z 324.076,A -85,B 0,C 180,E1 -2006.977,E2 -2006.977} C_VEL
LIN {X 0,Y 573.245,Z 324.073,A -85,B 0,C 180,E1 -2009.49,E2 -2009.49} C_VEL
LIN {X 0,Y 573.247,Z 324.078,A -85,B 0,C 180,E1 -2012.646,E2 -2012.646} C_VEL
LIN {X 0,Y 573.247,Z 324.073,A -85,B 0,C 180,E1 -2015.185,E2 -2015.185} C_VEL
LIN {X 0,Y 573.23,Z 324.078,A -85,B 0,C 180,E1 -2017.808,E2 -2017.808} C_VEL
LIN {X 0,Y 573.263,Z 324.076,A -85,B 0,C 180,E1 -2020.529,E2 -2020.529} C_VEL
LIN {X 0,Y 573.239,Z 324.076,A -85,B 0,C 180,E1 -2023.67,E2 -2023.67} C_VEL
LIN {X 0,Y 573.242,Z 324.076,A -85,B 0,C 180,E1 -2026.643,E2 -2026.643} C_VEL
LIN {X 0,Y 573.24,Z 324.075,A -85,B 0,C 180,E1 -2029.476,E2 -2029.476} C_VEL
LIN {X 0,Y 573.233,Z 324.083,A -85,B 0,C 180,E1 -2032.193,E2 -2032.193} C_VEL
LIN {X 0,Y 573.252,Z 324.073,A -85,B 0,C 180,E1 -2034.816,E2 -2034.816} C_VEL
LIN {X 0,Y 573.254,Z 324.073,A -85,B 0,C 180,E1 -2037.356,E2 -2037.356} C_VEL
LIN {X 0,Y 573.252,Z 324.074,A -85,B 0,C 180,E1 -2040.511,E2 -2040.511} C_VEL
LIN {X 0,Y 573.264,Z 324.071,A -85,B 0,C 180,E1 -2043.025,E2 -2043.025} C_VEL
LIN {X 0,Y 573.276,Z 324.072,A -85,B 0,C 180,E1 -2045.367,E2 -2045.367} C_VEL
LIN {X 0,Y 573.23,Z 324.077,A -85,B 0,C 180,E1 -2048.42,E2 -2048.42} C_VEL
LIN {X 0,Y 573.28,Z 324.069,A -85,B 0,C 180,E1 -2050.729,E2 -2050.729} C_VEL
LIN {X 0,Y 573.255,Z 324.08,A -85,B 0,C 180,E1 -2053.622,E2 -2053.622} C_VEL
LIN {X 0,Y 573.276,Z 324.079,A -85,B 0,C 180,E1 -2055.807,E2 -2055.807} C_VEL
LIN {X 0,Y 573.266,Z 324.071,A -85,B 0,C 180,E1 -2058.745,E2 -2058.745} C_VEL
LIN {X 0,Y 573.293,Z 324.075,A -85,B 0,C 180,E1 -2061.541,E2 -2061.541} C_VEL
LIN {X 0,Y 573.299,Z 324.067,A -85,B 0,C 180,E1 -2064.372,E2 -2064.372} C_VEL
LIN {X 0,Y 573.317,Z 324.069,A -85,B 0,C 180,E1 -2067.893,E2 -2067.893} C_VEL
LIN {X 0,Y 573.333,Z 324.063,A -85,B 0,C 180,E1 -2070.702,E2 -2070.702} C_VEL
LIN {X 0,Y 573.307,Z 324.066,A -85,B 0,C 180,E1 -2072.811,E2 -2072.811} C_VEL
LIN {X 0,Y 573.302,Z 324.073,A -85,B 0,C 180,E1 -2075.628,E2 -2075.628} C_VEL
LIN {X 0,Y 573.287,Z 324.068,A -85,B 0,C 180,E1 -2078.459,E2 -2078.459} C_VEL
LIN {X 0,Y 573.275,Z 324.079,A -85,B 0,C 180,E1 -2081.312,E2 -2081.312} C_VEL
LIN {X 0,Y 573.277,Z 324.07,A -85,B 0,C 180,E1 -2084.193,E2 -2084.193} C_VEL
LIN {X 0,Y 573.262,Z 324.078,A -85,B 0,C 180,E1 -2087.111,E2 -2087.111} C_VEL
LIN {X 0,Y 573.255,Z 324.072,A -85,B 0,C 180,E1 -2090.076,E2 -2090.076} C_VEL
LIN {X 0,Y 573.235,Z 324.083,A -85,B 0,C 180,E1 -2093.099,E2 -2093.099} C_VEL
LIN {X 0,Y 573.259,Z 324.078,A -85,B 0,C 180,E1 -2095.409,E2 -2095.409} C_VEL
LIN {X 0,Y 573.265,Z 324.071,A -85,B 0,C 180,E1 -2098.031,E2 -2098.031} C_VEL
LIN {X 0,Y 573.239,Z 324.08,A -85,B 0,C 180,E1 -2100.883,E2 -2100.883} C_VEL
LIN {X 0,Y 573.287,Z 324.071,A -85,B 0,C 180,E1 -2103.527,E2 -2103.527} C_VEL
LIN {X 0,Y 573.26,Z 324.071,A -85,B 0,C 180,E1 -2106.047,E2 -2106.047} C_VEL
LIN {X 0,Y 573.248,Z 324.078,A -85,B 0,C 180,E1 -2108.7,E2 -2108.7} C_VEL
LIN {X 0,Y 573.263,Z 324.073,A -85,B 0,C 180,E1 -2111.596,E2 -2111.596} C_VEL
LIN {X 0,Y 573.235,Z 324.077,A -85,B 0,C 180,E1 -2114.332,E2 -2114.332} C_VEL
LIN {X 0,Y 573.256,Z 324.078,A -85,B 0,C 180,E1 -2117.355,E2 -2117.355} C_VEL
LIN {X 0,Y 573.269,Z 324.12,A -85,B 0,C 180,E1 -2120.079,E2 -2120.079} C_VEL
LIN {X 0,Y 573.743,Z 326.998,A -85,B 0,C 180,E1 -2120.206,E2 -2120.206} C_VEL
LIN {X 0,Y 573.596,Z 339.576,A -85,B 0,C 180,E1 -2120.762,E2 -2120.762} C_VEL
LIN {X 0,Y 573.5,Z 351.075,A -85,B 0,C 180,E1 -2121.422,E2 -2121.422} C_VEL
LIN {X 0,Y 573.348,Z 361.827,A -85,B 0,C 180,E1 -2122.201,E2 -2122.201} C_VEL
LIN {X 0,Y 573.244,Z 371.559,A -85,B 0,C 180,E1 -2123.077,E2 -2123.077} C_VEL
LIN {X 0,Y 573.178,Z 380.178,A -85,B 0,C 180,E1 -2124.021,E2 -2124.021} C_VEL
LIN {X 0,Y 573.094,Z 387.754,A -85,B 0,C 180,E1 -2125.052,E2 -2125.052} C_VEL
LIN {X 0,Y 573.046,Z 393.898,A -85,B 0,C 180,E1 -2126.081,E2 -2126.081} C_VEL
LIN {X 0,Y 572.992,Z 398.016,A -85,B 0,C 180,E1 -2126.924,E2 -2126.924} C_VEL
LIN {X 0,Y 572.983,Z 401.59,A -85,B 0,C 180,E1 -2127.812,E2 -2127.812} C_VEL
LIN {X 0,Y 572.971,Z 405.176,A -85,B 0,C 180,E1 -2128.991,E2 -2128.991} C_VEL
LIN {X 0,Y 572.939,Z 406.946,A -85,B 0,C 180,E1 -2129.806,E2 -2129.806} C_VEL
LIN {X 0,Y 572.975,Z 408.143,A -85,B 0,C 180,E1 -2130.618,E2 -2130.618} C_VEL
LIN {X 0,Y 572.927,Z 408.813,A -85,B 0,C 180,E1 -2131.419,E2 -2131.419} C_VEL
LIN {X 0,Y 572.949,Z 408.97,A -85,B 0,C 180,E1 -2132.217,E2 -2132.217} C_VEL
LIN {X 0,Y 572.952,Z 408.047,A -85,B 0,C 180,E1 -2133.562,E2 -2133.562} C_VEL
LIN {X 0,Y 572.944,Z 406.399,A -85,B 0,C 180,E1 -2134.575,E2 -2134.575} C_VEL
LIN {X 0,Y 572.99,Z 403.429,A -85,B 0,C 180,E1 -2135.739,E2 -2135.739} C_VEL
LIN {X 0,Y 573.028,Z 399.181,A -85,B 0,C 180,E1 -2136.901,E2 -2136.901} C_VEL
LIN {X 0,Y 573.039,Z 393.762,A -85,B 0,C 180,E1 -2138.033,E2 -2138.033} C_VEL
LIN {X 0,Y 573.071,Z 388.295,A -85,B 0,C 180,E1 -2138.955,E2 -2138.955} C_VEL
LIN {X 0,Y 573.134,Z 381.372,A -85,B 0,C 180,E1 -2139.919,E2 -2139.919} C_VEL
LIN {X 0,Y 573.248,Z 372.302,A -85,B 0,C 180,E1 -2140.938,E2 -2140.938} C_VEL
LIN {X 0,Y 573.378,Z 363.068,A -85,B 0,C 180,E1 -2141.786,E2 -2141.786} C_VEL
LIN {X 0,Y 573.476,Z 351.83,A -85,B 0,C 180,E1 -2142.619,E2 -2142.619} C_VEL
LIN {X 0,Y 573.61,Z 340.766,A -85,B 0,C 180,E1 -2143.266,E2 -2143.266} C_VEL
LIN {X 0,Y 573.729,Z 328.715,A -85,B 0,C 180,E1 -2143.819,E2 -2143.819} C_VEL
LIN {X 0,Y 573.534,Z 325.35,A -85,B 0,C 180,E1 -2143.95,E2 -2143.95} C_VEL
LIN {X 0,Y 573.279,Z 324.232,A -85,B 0,C 180,E1 -2144.08,E2 -2144.08} C_VEL
LIN {X 0,Y 573.226,Z 324.078,A -85,B 0,C 180,E1 -2146.529,E2 -2146.529} C_VEL
LIN {X 0,Y 573.263,Z 324.081,A -85,B 0,C 180,E1 -2149.403,E2 -2149.403} C_VEL
LIN {X 0,Y 573.267,Z 324.072,A -85,B 0,C 180,E1 -2152.25,E2 -2152.25} C_VEL
LIN {X 0,Y 573.301,Z 324.073,A -85,B 0,C 180,E1 -2155.077,E2 -2155.077} C_VEL
LIN {X 0,Y 573.289,Z 324.07,A -85,B 0,C 180,E1 -2157.892,E2 -2157.892} C_VEL
LIN {X 0,Y 573.299,Z 324.068,A -85,B 0,C 180,E1 -2160,E2 -2160} C_VEL
LIN {X 0,Y 573.293,Z 324.071,A -85,B 0,C 180,E1 -2162.811,E2 -2162.811} C_VEL
LIN {X 0,Y 573.279,Z 324.073,A -85,B 0,C 180,E1 -2165.628,E2 -2165.628} C_VEL
LIN {X 0,Y 573.257,Z 324.074,A -85,B 0,C 180,E1 -2167.75,E2 -2167.75} C_VEL
LIN {X 0,Y 573.251,Z 324.075,A -85,B 0,C 180,E1 -2170.597,E2 -2170.597} C_VEL
LIN {X 0,Y 573.25,Z 324.077,A -85,B 0,C 180,E1 -2172.749,E2 -2172.749} C_VEL
LIN {X 0,Y 573.222,Z 324.084,A -85,B 0,C 180,E1 -2174.92,E2 -2174.92} C_VEL
LIN {X 0,Y 573.228,Z 324.076,A -85,B 0,C 180,E1 -2177.849,E2 -2177.849} C_VEL
LIN {X 0,Y 573.228,Z 324.076,A -85,B 0,C 180,E1 -2180.078,E2 -2180.078} C_VEL
LIN {X 0,Y 573.214,Z 324.079,A -85,B 0,C 180,E1 -2182.339,E2 -2182.339} C_VEL
LIN {X 0,Y 573.233,Z 324.078,A -85,B 0,C 180,E1 -2185.411,E2 -2185.411} C_VEL
LIN {X 0,Y 573.24,Z 324.074,A -85,B 0,C 180,E1 -2188.029,E2 -2188.029} C_VEL
LIN {X 0,Y 573.211,Z 324.087,A -85,B 0,C 180,E1 -2190.882,E2 -2190.882} C_VEL
LIN {X 0,Y 573.232,Z 324.077,A -85,B 0,C 180,E1 -2193.521,E2 -2193.521} C_VEL
LIN {X 0,Y 573.205,Z 324.079,A -85,B 0,C 180,E1 -2196.052,E2 -2196.052} C_VEL
LIN {X 0,Y 573.226,Z 324.085,A -85,B 0,C 180,E1 -2198.703,E2 -2198.703} C_VEL
LIN {X 0,Y 573.196,Z 324.08,A -85,B 0,C 180,E1 -2201.591,E2 -2201.591} C_VEL
LIN {X 0,Y 573.209,Z 324.083,A -85,B 0,C 180,E1 -2204.336,E2 -2204.336} C_VEL
LIN {X 0,Y 573.221,Z 324.086,A -85,B 0,C 180,E1 -2206.641,E2 -2206.641} C_VEL
LIN {X 0,Y 573.24,Z 324.076,A -85,B 0,C 180,E1 -2209.476,E2 -2209.476} C_VEL
LIN {X 0,Y 573.217,Z 324.084,A -85,B 0,C 180,E1 -2212.192,E2 -2212.192} C_VEL
LIN {X 0,Y 573.244,Z 324.221,A -85,B 0,C 180,E1 -2213.68,E2 -2213.68} C_VEL
LIN {X 0,Y 573.897,Z 328.68,A -85,B 0,C 180,E1 -2214.65,E2 -2214.65} C_VEL
LIN {X 0,Y 573.66,Z 342.472,A -85,B 0,C 180,E1 -2217.382,E2 -2217.382} C_VEL
LIN {X 0,Y 573.792,Z 357.153,A -85,B 0,C 180,E1 -2220.177,E2 -2220.177} C_VEL
LIN {X 0,Y 573.811,Z 371.686,A -85,B 0,C 180,E1 -2222.856,E2 -2222.856} C_VEL
LIN {X 0,Y 573.835,Z 383.457,A -85,B 0,C 180,E1 -2225.001,E2 -2225.001} C_VEL
LIN {X 0,Y 573.678,Z 397.192,A -85,B 0,C 180,E1 -2227.681,E2 -2227.681} C_VEL
LIN {X 0,Y 573.498,Z 412.843,A -85,B 0,C 180,E1 -2230.679,E2 -2230.679} C_VEL
LIN {X 0,Y 573.355,Z 426.696,A -85,B 0,C 180,E1 -2233.289,E2 -2233.289} C_VEL
LIN {X 0,Y 573.253,Z 442.189,A -85,B 0,C 180,E1 -2236.169,E2 -2236.169} C_VEL
LIN {X 0,Y 573.191,Z 449.053,A -85,B 0,C 180,E1 -2237.408,E2 -2237.408} C_VEL
LIN {X 0,Y 573.417,Z 450.752,A -85,B 0,C 180,E1 -2237.48,E2 -2237.48} C_VEL
LIN {X 0,Y 573.856,Z 454.932,A -85,B 0,C 180,E1 -2237.557,E2 -2237.557} C_VEL
LIN {X 0,Y 573.786,Z 467.523,A -85,B 0,C 180,E1 -2237.847,E2 -2237.847} C_VEL
LIN {X 0,Y 573.67,Z 480.363,A -85,B 0,C 180,E1 -2238.294,E2 -2238.294} C_VEL
LIN {X 0,Y 573.593,Z 492.936,A -85,B 0,C 180,E1 -2238.89,E2 -2238.89} C_VEL
LIN {X 0,Y 573.442,Z 504.211,A -85,B 0,C 180,E1 -2239.585,E2 -2239.585} C_VEL
LIN {X 0,Y 573.334,Z 514.592,A -85,B 0,C 180,E1 -2240.386,E2 -2240.386} C_VEL
LIN {X 0,Y 573.237,Z 523.101,A -85,B 0,C 180,E1 -2241.185,E2 -2241.185} C_VEL
LIN {X 0,Y 573.16,Z 530.95,A -85,B 0,C 180,E1 -2242.071,E2 -2242.071} C_VEL
LIN {X 0,Y 573.076,Z 538.94,A -85,B 0,C 180,E1 -2243.182,E2 -2243.182} C_VEL
LIN {X 0,Y 573.069,Z 545.677,A -85,B 0,C 180,E1 -2244.37,E2 -2244.37} C_VEL
LIN {X 0,Y 573.028,Z 550.368,A -85,B 0,C 180,E1 -2245.428,E2 -2245.428} C_VEL
LIN {X 0,Y 573.022,Z 553.955,A -85,B 0,C 180,E1 -2246.484,E2 -2246.484} C_VEL
LIN {X 0,Y 572.959,Z 555.807,A -85,B 0,C 180,E1 -2247.188,E2 -2247.188} C_VEL
LIN {X 0,Y 572.94,Z 557.201,A -85,B 0,C 180,E1 -2247.891,E2 -2247.891} C_VEL
LIN {X 0,Y 572.941,Z 558.784,A -85,B 0,C 180,E1 -2249.297,E2 -2249.297} C_VEL
LIN {X 0,Y 572.938,Z 559,A -85,B 0,C 180,E1 -2250,E2 -2250} C_VEL
LIN {X 0,Y 572.946,Z 558.187,A -85,B 0,C 180,E1 -2251.406,E2 -2251.406} C_VEL
LIN {X 0,Y 572.94,Z 557.202,A -85,B 0,C 180,E1 -2252.109,E2 -2252.109} C_VEL
LIN {X 0,Y 572.959,Z 555.808,A -85,B 0,C 180,E1 -2252.812,E2 -2252.812} C_VEL
LIN {X 0,Y 573.014,Z 552.898,A -85,B 0,C 180,E1 -2253.868,E2 -2253.868} C_VEL
LIN {X 0,Y 572.962,Z 548.955,A -85,B 0,C 180,E1 -2254.926,E2 -2254.926} C_VEL
LIN {X 0,Y 573.074,Z 543.869,A -85,B 0,C 180,E1 -2255.983,E2 -2255.983} C_VEL
LIN {X 0,Y 573.104,Z 537.46,A -85,B 0,C 180,E1 -2257.044,E2 -2257.044} C_VEL
LIN {X 0,Y 573.174,Z 529.481,A -85,B 0,C 180,E1 -2258.106,E2 -2258.106} C_VEL
LIN {X 0,Y 573.254,Z 521.345,A -85,B 0,C 180,E1 -2258.993,E2 -2258.993} C_VEL
LIN {X 0,Y 573.351,Z 511.396,A -85,B 0,C 180,E1 -2259.881,E2 -2259.881} C_VEL
LIN {X 0,Y 573.499,Z 500.191,A -85,B 0,C 180,E1 -2260.68,E2 -2260.68} C_VEL
LIN {X 0,Y 573.628,Z 489.199,A -85,B 0,C 180,E1 -2261.305,E2 -2261.305} C_VEL
LIN {X 0,Y 573.692,Z 476.99,A -85,B 0,C 180,E1 -2261.84,E2 -2261.84} C_VEL
LIN {X 0,Y 573.809,Z 464.161,A -85,B 0,C 180,E1 -2262.242,E2 -2262.242} C_VEL
LIN {X 0,Y 573.66,Z 452.324,A -85,B 0,C 180,E1 -2262.489,E2 -2262.489} C_VEL
LIN {X 0,Y 573.22,Z 449.314,A -85,B 0,C 180,E1 -2262.569,E2 -2262.569} C_VEL
LIN {X 0,Y 573.222,Z 444.145,A -85,B 0,C 180,E1 -2263.47,E2 -2263.47} C_VEL
LIN {X 0,Y 573.333,Z 428.494,A -85,B 0,C 180,E1 -2266.375,E2 -2266.375} C_VEL
LIN {X 0,Y 573.468,Z 414.799,A -85,B 0,C 180,E1 -2268.951,E2 -2268.951} C_VEL
LIN {X 0,Y 573.635,Z 401.105,A -85,B 0,C 180,E1 -2271.564,E2 -2271.564} C_VEL
LIN {X 0,Y 573.817,Z 385.454,A -85,B 0,C 180,E1 -2274.608,E2 -2274.608} C_VEL
LIN {X 0,Y 573.868,Z 372.085,A -85,B 0,C 180,E1 -2277.141,E2 -2277.141} C_VEL
LIN {X 0,Y 573.916,Z 358.037,A -85,B 0,C 180,E1 -2279.827,E2 -2279.827} C_VEL
LIN {X 0,Y 573.937,Z 343.002,A -85,B 0,C 180,E1 -2282.809,E2 -2282.809} C_VEL
LIN {X 0,Y 574.204,Z 330.747,A -85,B 0,C 180,E1 -2285.331,E2 -2285.331} C_VEL
LIN {X 0,Y 573.55,Z 325.611,A -85,B 0,C 180,E1 -2286.461,E2 -2286.461} C_VEL
LIN {X 0,Y 573.236,Z 324.183,A -85,B 0,C 180,E1 -2286.813,E2 -2286.813} C_VEL
LIN {X 0,Y 573.225,Z 324.086,A -85,B 0,C 180,E1 -2289.608,E2 -2289.608} C_VEL
LIN {X 0,Y 573.212,Z 324.079,A -85,B 0,C 180,E1 -2292.638,E2 -2292.638} C_VEL
LIN {X 0,Y 573.2,Z 324.088,A -85,B 0,C 180,E1 -2295.326,E2 -2295.326} C_VEL
LIN {X 0,Y 573.231,Z 324.082,A -85,B 0,C 180,E1 -2297.599,E2 -2297.599} C_VEL
LIN {X 0,Y 573.229,Z 324.076,A -85,B 0,C 180,E1 -2300.568,E2 -2300.568} C_VEL
